(* Logix 5000 project; controller P2 vendor 1 type 14 code 92 rev 20.55; software revision 20.01 *)

TASK MainTask (continuous, watchdog 500 ms) : MainProgram

MODULES
   Local : vendor 1 type 14 code 92 (ICP 0, rev 20.55)
      P2_EN2T_PCN : 1756-EN2T (ICP 1, Ethernet 192.168.1.20, rev 10.1)
         P5 : 1756-EN2T (Ethernet 192.168.1.50, rev 10.1, Output RPI 10 ms)
            P5_CONTROLLER : vendor 1 type 14 code 92 (ICP 0, rev 20.1)
         P4 : 1756-EN2T (Ethernet 192.168.1.40, rev 10.1, Output RPI 10 ms)
            P4_CONTROLLER : vendor 1 type 14 code 92 (ICP 0, rev 20.1)
         P3 : 1756-EN2T (Ethernet 192.168.1.30, rev 10.1, Output RPI 10 ms)
            P3_CONTROLLER : vendor 1 type 14 code 92 (ICP 0, rev 20.1)
      P2_EN2TR_RIO : vendor 1 type 12 code 200 (ICP 2, Ethernet 192.168.0.20, rev 10.1)
         RIO2 : 1794-AENTR (Ethernet 192.168.0.22, rev 1.1, Output RPI 20 ms)
            RIO2_DI : 1794-IB32 (Flex 0, rev 1.1, Input RPI 20 ms)
            RIO2_DO : vendor 1 type 7 code 35 (Flex 1, rev 1.1)
            RIO2_AI : 1794-IE12 (Flex 2, rev 1.1, Output RPI 80 ms)
         WRIO2 : vendor 309 type 12 code 1000 (Ethernet 192.168.0.25, rev 3.1, Output RPI 20 ms)
            WRIO2_AI : 1734-IE4C (PointIO 1, rev 3.1, Input RPI 80 ms)
END_MODULES

TYPE AIN_UDT :
STRUCT
   Pv : REAL;
   Heu : REAL;
   Leu : REAL;
   SAHH : REAL;
   SAH : REAL;
   SAL : REAL;
   SALL : REAL;
   AHH : BOOL;
   AH : BOOL;
   AL : BOOL;
   ALL : BOOL;
   Wifi_Enb : BOOL;
   Hty : BOOL;
   Sim : BOOL;
   Sim_PV : REAL;
END_STRUCT
END_TYPE

TYPE AUTOINP_UDT :
STRUCT
   ON : BOOL;
END_STRUCT
END_TYPE

TYPE ControllerLEDStatus :
STRUCT
   Off : BOOL;
   SolidGreen : BOOL;
   FlashingGreen : BOOL;
   SolidYellow : BOOL;
   FlashingYellow : BOOL;
   FlashingRed : BOOL;
   SolidRed : BOOL;
END_STRUCT
END_TYPE

TYPE DOSING_SETPOINT_UDT :
STRUCT
   High_Setpoint : REAL;
   Low_Setpoint : REAL;
END_STRUCT
END_TYPE

TYPE Duty2_UDT :
STRUCT
   Selection : INT;
   Pmp1_Not_Avl : BOOL;
   Pmp2_Not_Avl : BOOL;
   Selected_Pmp_Not_Avl : BOOL;
   Both_Pmp_Not_Avl : BOOL;
END_STRUCT
END_TYPE

TYPE FaultRecord :
STRUCT
   timelow : DINT;
   timehigh : DINT;
   type : INT;
   code : INT;
   info : DINT[8];
END_STRUCT
END_TYPE

TYPE FIT_UDT :
STRUCT
   Pv : REAL;
   Heu : REAL;
   Leu : REAL;
   SAHH : REAL;
   SAH : REAL;
   SAL : REAL;
   SALL : REAL;
   Totaliser : REAL;
   AHH : BOOL;
   AH : BOOL;
   AL : BOOL;
   ALL : BOOL;
   Sim : BOOL;
   Sim_PV : REAL;
   Wifi_Enb : BOOL;
   Rst_Totaliser : BOOL;
   Hty : BOOL;
END_STRUCT
END_TYPE

TYPE Logix_Status_FP :
STRUCT
   ClearMinorFaults : DINT;
   Sts_MinorFaultEvents : DINT;
   Sts_MinorFaultBits : DINT;
   Sts_Redundant : DINT;
   Set_FaceplateAnimation : DINT;
   Val_ProductCode : DINT;
   MemoryTemp : INT[29];
   Val_raw_data : INT;
   Sts_IO_LED_raw : INT;
   Sts_ProductCode : INT;
   Val_Force_data_raw : INT;
   MemoryRequestData : SINT[12];
   Sts_Force_Installed : BOOL;
   Sts_Force_Enabled : BOOL;
   Sts_Faulted : BOOL;
   Sts_Run : BOOL;
   Sts_Program : BOOL;
   Sts_Minor_fault : BOOL;
   Sts_Major_fault : BOOL;
   Sts_KS_in_run : BOOL;
   Sts_KS_in_program : BOOL;
   Sts_KS_in_remote : BOOL;
   Sts_Changingmodes : BOOL;
   Sts_Test : BOOL;
   Sts_Ladder_Working : BOOL;
   Cmd_ClearFaultRecord : BOOL;
   Set_Controller_Description : STRING;
   UpdateDelayTimer : TIMER;
   Val_MajorFault : FaultRecord;
   Val_MFS : FaultRecord;
   Sts_IO_LED : ControllerLEDStatus;
   Sts_Battery_LED : ControllerLEDStatus;
   MemoryData : Memory_Data;
   TEST : DINT;
END_STRUCT
END_TYPE

TYPE Memory_Data :
STRUCT
   Free_Mem_IO : DINT;
   Free_Mem_DT : DINT;
   Free_Memory : DINT;
   Total_Mem_IO : DINT;
   Total_Mem_DT : DINT;
   Total_Memory : DINT;
   Biggest_IO_Mem_Size_Ava : DINT;
   Biggest_DT_Mem_Size_Ava : DINT;
END_STRUCT
END_TYPE

TYPE MV_UDT :
STRUCT
   Cmd : INT;
   Status : INT;
   Reset : BOOL;
   Auto : BOOL;
   FTO : BOOL;
   FTC : BOOL;
   Avl : BOOL;
END_STRUCT
END_TYPE

TYPE PLANT_AUTO_UDT :
STRUCT
   ON : BOOL;
   OFF : BOOL;
END_STRUCT
END_TYPE

TYPE PLANT_UDT :
STRUCT
   START : BOOL;
   STOP : BOOL;
END_STRUCT
END_TYPE

TYPE PMP_UDT :
STRUCT
   Cmd : INT;
   Status : INT;
   RunMin : REAL;
   Total_RunMin : REAL;
   RunHr : REAL;
   Total_RunHr : REAL;
   Remote : BOOL;
   Auto : BOOL;
   Fault : BOOL;
   Avl : BOOL;
   Permissive : DINT;
   Shutdown : DINT;
   SD : DINT;
   Reset : BOOL;
   Reset_RunHr : BOOL;
   FTR : BOOL;
   FTS : BOOL;
END_STRUCT
END_TYPE

TYPE PRECONDITION_UDT :
STRUCT
   PERMISSIVE1 : BOOL;
   PERMISSIVE2 : BOOL;
   PERMISSIVE3 : BOOL;
   PERMISSIVE4 : BOOL;
   PERMISSIVE5 : BOOL;
   SHUTDOWN1 : BOOL;
   SHUTDOWN2 : BOOL;
   SHUTDOWN3 : BOOL;
   SHUTDOWN4 : BOOL;
   SHUTDOWN5 : BOOL;
END_STRUCT
END_TYPE

TYPE RED_STAT :
STRUCT
   Redundancy_status_of_the_controller : INT;
   Redundancy_state_of_the_partner : INT;
END_STRUCT
END_TYPE

TYPE SWITCH_UDT :
STRUCT
   Alarm : BOOL;
   Delay : DINT;
END_STRUCT
END_TYPE

TYPE WIFI_UDT :
STRUCT
   PLC_WIFI : BOOL;
   RIO_WIFI : BOOL;
END_STRUCT
END_TYPE

ADD_ON_INSTRUCTION AIN_FBD   (* revision 1.0 *)
VAR_INPUT
   WRIO_Enb : BOOL; {visible}
   Raw_RIO : INT; {visible}
   Raw_WRIO : INT; {visible}
   L_Raw_RIO : INT; {visible}
   H_Raw_RIO : INT; {visible}
   L_Raw_WRIO : INT; {visible}
   H_Raw_WRIO : INT; {visible}
   HEU : INT; {visible}
   LEU : INT; {visible}
END_VAR
VAR_OUTPUT
   Hty : BOOL; {visible}
   Wifi_Enb : BOOL; {access Read Only, visible}
   AHH : BOOL; {visible}
   AH : BOOL; {access Read Only, visible}
   AL : BOOL; {access Read Only, visible}
   ALL : BOOL; {visible}
END_VAR
VAR_INPUT
   SAHH : REAL; {visible}
   SAH : REAL; {visible}
   SAL : REAL; {visible}
   SALL : REAL; {visible}
   Simulation : BOOL; {visible}
   RIO_Hty : BOOL; {visible}
   WRIO_Hty : BOOL; {visible}
END_VAR
VAR_IN_OUT
   Pv : REAL; {required}
   Sim_PV : REAL; {required}
   HMI : AIN_UDT; {required}
END_VAR
VAR
   SCALE : SCALE; {access None}
   ALM : ALARM; {access None}
   _Raw : INT; {access None}
   _L_Raw : INT; {access None}
   _H_Raw : INT; {access None}
   _Inst_Hty : BOOL; {access None}
END_VAR

ROUTINE Logic   (* structured text *)
   (*RIO and Wireless RIO Selection*)
   
   IF WRIO_Enb THEN
   	Wifi_Enb	:= 1;
   	_Raw		:= Raw_WRIO;
   	_H_Raw		:= H_Raw_WRIO;
   	_L_Raw		:= L_Raw_WRIO;
   	_Inst_Hty 	:= WRIO_Hty;
   ELSE
   	Wifi_Enb	:= 0;
   	_Raw		:= Raw_RIO;
   	_H_Raw		:= H_Raw_RIO;
   	_L_Raw		:= L_Raw_RIO;
   	_Inst_Hty 	:= RIO_Hty;
   END_IF;
   
   (*Calculation for PV*)
   IF Simulation THEN
   	Pv	:=Sim_PV;
   ELSE
   	SCALE.In		:=_Raw;
   	SCALE.InRawMax	:=_H_Raw;
   	SCALE.InRawMin	:=_L_Raw;
   	SCALE.InEUMax	:=HEU;
   	SCALE.InEUMin	:=LEU;
   	SCL(SCALE);
   
   	IF SCALE.Out<0 THEN
   		Pv	:= 0.0;
   	ELSE
   		Pv	:=SCALE.Out;
   	END_IF;
   
   	Sim_PV	:=Pv;
   
   END_IF;
   
   (*Alarms*)
   ALM.In			:=Pv;
   ALM.HHLimit		:=SAHH;
   ALM.HLimit		:=SAH;
   ALM.LLimit		:=SAL;
   ALM.LLLimit		:=SALL;
   ALM(ALM);
   
   AHH				:=ALM.HHAlarm;
   AH				:=ALM.HAlarm;
   AL				:=ALM.LAlarm;
   ALL				:=ALM.LLAlarm;
   
   Hty:= _Inst_Hty AND (_Raw > _L_Raw) AND (_Raw < _H_Raw)  ;
   
   
   
   
   
   
END_ROUTINE
END_ADD_ON_INSTRUCTION

ADD_ON_INSTRUCTION Duty2_FBD   (* revision 1.0 *)
VAR_INPUT
   AutoInp : BOOL; {visible}
   Selection : INT; {visible}
   Pmp1_Avl : BOOL; {visible}
   Pmp2_Avl : BOOL; {visible}
END_VAR
VAR_OUTPUT
   Start_Pmp1 : BOOL; {visible}
   Start_Pmp2 : BOOL; {visible}
END_VAR
VAR_IN_OUT
   HMI : Duty2_UDT; {required}
END_VAR

ROUTINE Logic   (* structured text *)
   IF AutoInp THEN
   	CASE Selection OF
   		(*PUMP 1 *)
   		1:
   			IF Pmp1_Avl THEN
   				Start_Pmp1					:=1;
   				Start_Pmp2					:=0;
   				HMI.Selected_Pmp_Not_Avl	:=0;
   			ELSIF NOT Pmp1_Avl AND Pmp2_Avl THEN
   				Start_Pmp1					:=0;
   				Start_Pmp2					:=1;
   				HMI.Selected_Pmp_Not_Avl	:=1;
   			ELSIF NOT Pmp1_Avl AND NOT Pmp2_Avl	THEN
   				Start_Pmp1					:=0;
   				Start_Pmp2					:=0;
   			END_IF;
   
   		(*PUMP 2 *)
   		2:
   			IF Pmp2_Avl THEN
   				Start_Pmp1					:=0;
   				Start_Pmp2					:=1;
   				HMI.Selected_Pmp_Not_Avl	:=0;
   			ELSIF NOT Pmp2_Avl AND Pmp1_Avl THEN
   				Start_Pmp1					:=1;
   				Start_Pmp2					:=0;
   				HMI.Selected_Pmp_Not_Avl	:=1;
   			ELSIF NOT Pmp1_Avl AND NOT Pmp2_Avl	THEN
   				Start_Pmp1					:=0;
   				Start_Pmp2					:=0;
   			END_IF;
   	END_CASE;
   ELSE
   	Start_Pmp1					:=0;
   	Start_Pmp2					:=0;
   END_IF;
   
   
END_ROUTINE
END_ADD_ON_INSTRUCTION

ADD_ON_INSTRUCTION FIT_FBD   (* revision 1.0 *)
VAR_INPUT
   WRIO_Enb : BOOL; {visible}
   Raw_RIO : INT; {visible}
   Raw_WRIO : INT; {visible}
   L_Raw_RIO : INT; {visible}
   H_Raw_RIO : INT; {visible}
   L_Raw_WRIO : INT; {visible}
   H_Raw_WRIO : INT; {visible}
   HEU : REAL; {visible}
   LEU : REAL; {visible}
END_VAR
VAR_OUTPUT
   Hty : BOOL; {visible}
   Wifi_Enb : BOOL; {visible}
   AHH : BOOL; {visible}
   AH : BOOL; {access Read Only, visible}
   AL : BOOL; {access Read Only, visible}
   ALL : BOOL; {visible}
END_VAR
VAR_INPUT
   SAHH : REAL; {visible}
   SAH : REAL; {visible}
   SAL : REAL; {visible}
   SALL : REAL; {visible}
   Simulation : BOOL; {visible}
   RIO_Hty : BOOL; {visible}
   WRIO_Hty : BOOL; {visible}
   Totaliser_Enb : BOOL; {visible}
   Rst_Totaliser : BOOL; {visible}
END_VAR
VAR_IN_OUT
   Totaliser : REAL; {required}
   Pv : REAL; {required}
   Sim_Pv : REAL; {required}
   HMI : FIT_UDT; {required}
END_VAR
VAR
   SCALE : SCALE; {access None}
   ALM : ALARM; {access None}
   TON : FBD_TIMER; {access None}
   _SEC_P : BOOL; {access None}
   _Inst_Hty : BOOL; {access None}
   _L_Raw : INT; {access None}
   _H_Raw : INT; {access None}
   _Raw : INT; {access None}
   R_TRIG : FBD_ONESHOT; {access None}
END_VAR

ROUTINE Logic   (* structured text *)
   (*RIO and Wireless RIO Selection*)
   
   IF WRIO_Enb THEN
   	Wifi_Enb	:= 1;
   	_Raw		:= Raw_WRIO;
   	_H_Raw		:= H_Raw_WRIO;
   	_L_Raw		:= L_Raw_WRIO;
   	_Inst_Hty 	:= WRIO_Hty;
   ELSE
   	Wifi_Enb	:= 0;
   	_Raw		:= Raw_RIO;
   	_H_Raw		:= H_Raw_RIO;
   	_L_Raw		:= L_Raw_RIO;
   	_Inst_Hty 	:= RIO_Hty;
   END_IF;
   
   (*Calculation for PV*)
   IF Simulation THEN
   	Pv	:= Sim_Pv   ;
   ELSE
   	SCALE.In		:=_Raw;
   	SCALE.InRawMax	:=_H_Raw;
   	SCALE.InRawMin	:=_L_Raw;
   	SCALE.InEUMax	:=HEU;
   	SCALE.InEUMin	:=LEU;
   	SCL(SCALE);
   	IF SCALE.Out>0 THEN
   		Pv	:=SCALE.Out;
   	ELSIF SCALE.Out<=0 THEN
   		Pv	:=0.0;
   	END_IF;
   
   	Sim_Pv	:=Pv;
   END_IF;
   
   (*Alarms*)
   ALM.In			:=Pv;
   ALM.HHLimit		:=SAHH;
   ALM.HLimit		:=SAH;
   ALM.LLimit		:=SAL;
   ALM.LLLimit		:=SALL;
   ALM(ALM);
   
   AHH				:=ALM.HHAlarm;
   AH				:=ALM.HAlarm;
   AL				:=ALM.LAlarm;
   ALL				:=ALM.LLAlarm;
   
   (*SECOND PULSE*)
   TON.PRE	:=1000;
   TON.TimerEnable	:=1;
   TONR(TON );
   R_TRIG.InputBit :=TON.DN ;
   OSRI( R_TRIG);
   _SEC_P  := R_TRIG.OutputBit;
   TON.Reset := _SEC_P;
   
   IF Totaliser_Enb THEN
   	IF _SEC_P THEN
   		HMI.Totaliser := HMI.Totaliser +  (ABS(Pv) / 3600 );
   	END_IF;
   END_IF;
   
   IF  Rst_Totaliser   THEN
   	HMI.Totaliser	:=0;
   END_IF;
   
   Hty:= _Inst_Hty AND (_Raw > _L_Raw) AND (_Raw < _H_Raw)  ;
   
   
   
   
   
   
END_ROUTINE
END_ADD_ON_INSTRUCTION

ADD_ON_INSTRUCTION MV_FBD   (* revision 1.0 *)
VAR_INPUT
   Auto : BOOL; {visible}
END_VAR
VAR_OUTPUT
   Cmd_Open : BOOL; {visible}
   Cmd_Close : BOOL; {visible}
   FTO : BOOL; {visible}
   FTC : BOOL; {access Read Only, visible}
END_VAR
VAR_INPUT
   AutoInp : BOOL; {visible}
   ZSO : BOOL; {visible}
   Open_TM : DINT; {visible}
   ZSC : BOOL; {visible}
   Close_TM : DINT; {visible}
END_VAR
VAR_IN_OUT
   Cmd : INT; {required}
   HMI : MV_UDT; {required}
END_VAR
VAR
   TON_Open_TM : FBD_TIMER; {access None}
   TON_Close_TM : FBD_TIMER; {access None}
END_VAR

ROUTINE Logic   (* structured text *)
   (*Fail to Close*)
   TON_Close_TM.PRE 			:= 	Close_TM*1000;
   TON_Close_TM.TimerEnable 	:=  Cmd_Close;
   TONR(TON_Close_TM);
   
   (*Fail to Open*)
   TON_Open_TM.PRE 			:= 	Open_TM*1000;
   TON_Open_TM.TimerEnable 	:= 	Cmd_Open;
   TONR(TON_Open_TM);
   
   IF ZSC THEN
   	HMI.Status	:=1;
   ELSIF ZSO THEN
   	HMI.Status	:=2;
   ELSE
   	HMI.Status	:=0;
   END_IF;
   
   HMI.Avl:= Auto AND NOT FTC AND NOT FTO;
   
   IF HMI.Reset THEN
   	(*IF NOT TON_Close_TM.DN AND ZSC THEN*)
   			FTC		:= 0;
   	(*END_IF;*)
   	(*IF NOT TON_Open_TM.DN AND ZSO THEN*)
   			FTO		:= 0;
   	(*END_IF;*)
   END_IF;
   
   IF  NOT Auto THEN
   	CASE HMI.Cmd OF
   		1:	(*CLOSE*)
   			Cmd_Close	:= 1;
   			Cmd_Open	:= 0;
   			IF TON_Close_TM.DN AND (NOT ZSC) THEN
   				FTC		:= 1;
   				FTO		:= 0;
   			END_IF;
   		2:	(*OPEN*)
   			IF FTO OR FTC    THEN
   				HMI.Cmd := 1;
   			END_IF;
   
   			IF NOT FTC AND NOT FTO THEN
   				Cmd_Close	:= 0;
   				Cmd_Open	:= 1;
   			END_IF;
   
   			IF TON_Open_TM.DN AND (NOT ZSO) THEN
   				FTC		:= 0;
   				FTO		:= 1;
   				HMI.Cmd := 1;
   			END_IF;
   	END_CASE;
   ELSE
   	(*Maintain Last status when switching from Auto to Manual*)
   	IF ZSO THEN
   		Cmd	:= 2;
   	END_IF;
   	IF ZSC THEN
   		Cmd	:= 1;
   	END_IF;
   
   	IF  AutoInp AND (NOT FTC AND NOT FTO) THEN
   		Cmd_Close	:= 0;
   		Cmd_Open	:= 1;
   		IF TON_Open_TM.DN AND (NOT ZSO) THEN
   			FTC		:= 0;
   			FTO		:= 1;
   		END_IF;
   	ELSE
   		Cmd_Close	:= 1;
   		Cmd_Open	:= 0;
   		IF TON_Close_TM.DN AND (NOT ZSC) THEN
   			FTC		:= 1;
   			FTO		:= 0;
   		END_IF;
   	END_IF;
   END_IF;
   
   
END_ROUTINE
END_ADD_ON_INSTRUCTION

ADD_ON_INSTRUCTION PMP_FBD   (* revision 1.0 *)
VAR_OUTPUT
   Cmd_Start : BOOL; {visible}
   Avl : BOOL; {visible}
   Fault : BOOL; {visible}
   FT_Stop : BOOL; {visible}
   FT_Start : BOOL; {visible}
   RunHr : REAL; {visible}
   Total_RunHr : REAL; {visible}
   SD : DINT; {access Read Only, visible}
END_VAR
VAR_INPUT
   Auto : BOOL; {visible}
   AutoInp : BOOL; {visible}
   Remote : BOOL; {visible}
   Run : BOOL; {visible}
   Trip : BOOL; {visible}
   Start_TM : DINT; {visible}
   Stop_TM : DINT; {visible}
   Rst : BOOL; {visible}
   Rst_RunHr : BOOL; {visible}
   Permissive : DINT; {visible}
   Shutdown : DINT; {visible}
END_VAR
VAR_IN_OUT
   RunMin : REAL; {required}
   Total_RunMin : REAL; {required}
   Cmd : INT; {required}
   HMI : PMP_UDT; {required}
END_VAR
VAR
   TON_Start_TM : FBD_TIMER; {access None}
   TON_Stop_TM : FBD_TIMER; {access None}
   _Min_P : BOOL; {access None}
   TON_Min : FBD_TIMER; {access None}
   R_TRIG_SEC : FBD_ONESHOT; {access None}
END_VAR

ROUTINE Logic   (* structured text *)
   (*Fail to Start*)
   TON_Start_TM.PRE 			:= 	Start_TM*1000;
   TON_Start_TM.TimerEnable 	:=  Cmd_Start;
   TONR(TON_Start_TM);
   
   (*Fail to Stop*)
   TON_Stop_TM.PRE 			:= 	Stop_TM*1000;
   TON_Stop_TM.TimerEnable 	:=  NOT Cmd_Start;
   TONR(TON_Stop_TM);
   
   IF (NOT Run) THEN
   	HMI.Status	:=1;
   ELSE
   	HMI.Status	:=2;
   END_IF;
   
   IF Fault THEN
   	HMI.Fault:= 1;
   ELSE
   	HMI.Fault:= 0;
   END_IF;
   
   IF HMI.Reset THEN
   	IF NOT TON_Stop_TM.DN THEN
   			FT_Stop		:= 0;
   	END_IF;
   	IF NOT TON_Start_TM.DN THEN
   			FT_Start	:= 0;
   	END_IF;
   
   	SD :=0;
   
   END_IF;
   
   Fault		:=Trip OR SD<>0;
   HMI.Remote	:=Remote;
   Avl:= Auto AND Remote AND NOT Fault AND NOT FT_Start AND NOT FT_Stop AND SD=0 ;
   
   IF Remote THEN
   	IF  NOT Auto THEN
   		CASE HMI.Cmd OF
   			1:	(*Stop*)
   				Cmd_Start	:=0;
   				IF TON_Stop_TM.DN AND Run THEN
   					FT_Start	:= 0;
   					FT_Stop		:= 1;
   				END_IF;
   			2:	(*OPEN*)
   				IF NOT Fault AND NOT FT_Start AND NOT FT_Stop AND (Permissive=-1) AND HMI.SD=0 THEN
   					Cmd_Start	:= 1;
   				ELSIF Cmd_Start AND (HMI.SD<>0) OR Fault THEN
   					SD				:= HMI.SD;
   					Cmd_Start		:= 0;
   					HMI.Cmd 		:= 1;
   				ELSIF (Permissive<>-1) THEN
   					HMI.Cmd 		:= 1;
   				END_IF;
   
   				IF TON_Start_TM.DN AND NOT Run THEN
   					FT_Start	:= 1;
   					FT_Stop		:= 0;
   					Cmd_Start	:= 0;
   					HMI.Cmd 	:= 1;
   				END_IF;
   		END_CASE;
   	ELSE
   		IF Run THEN
   			Cmd	:= 2;
   		END_IF;
   		IF (NOT Run) OR Fault OR FT_Start OR FT_Stop THEN
   			Cmd	:= 1;
   		END_IF;
   
   		IF  AutoInp  THEN
   			IF NOT Fault AND NOT FT_Start AND NOT FT_Stop AND (Permissive=-1) AND HMI.SD=0  THEN
   				Cmd_Start	:=1;
   			ELSIF Cmd_Start OR (HMI.SD<>0) OR Fault THEN
   				SD			:= HMI.SD;
   				Cmd_Start	:=0;
   			END_IF;
   
   			IF TON_Start_TM.DN AND NOT Run THEN
   				FT_Start	:= 1;
   				FT_Stop		:= 0;
   				Cmd_Start	:= 0;
   				HMI.Cmd 	:= 1;
   			END_IF;
   		ELSE
   			Cmd_Start	:=0;
   			IF TON_Stop_TM.DN AND Run THEN
   				FT_Start	:= 0;
   				FT_Stop		:= 1;
   
   			END_IF;
   		END_IF;
   	END_IF;
   
   ELSE (*Local*)
   	Cmd_Start	:=0;
   	Cmd	:= 1;
   
   	FT_Start	:= 0;
   	FT_Stop		:= 0;
   
   
   
   
   	(*	IF Run THEN
   			Cmd	:= 2;
   		END_IF;
   		IF (NOT Run) OR Fault OR FT_Start OR FT_Stop THEN
   			Cmd	:= 1;
   		END_IF;
   		*)
   END_IF;
   
   (*1 MIN PULSE*)
   TON_Min.PRE	:=60000;
   TON_Min.TimerEnable	:=1;
   TONR(TON_Min );
   R_TRIG_SEC.InputBit :=TON_Min.DN ;
   OSRI( R_TRIG_SEC);
   _Min_P  := R_TRIG_SEC.OutputBit;
   TON_Min.Reset 	:= _Min_P;
   
   IF Run THEN
   	IF _Min_P THEN
   		RunMin 			:=RunMin + 1.0;
   		Total_RunMin	:=Total_RunMin + 1.0;
   	END_IF;
   END_IF;
   
   RunHr 				:=RunMin/60.0;
   Total_RunHr			:=Total_RunMin/60.0;
   
   IF  Rst_RunHr THEN
   	RunMin	:=0;
   END_IF;
   
   
   
END_ROUTINE
END_ADD_ON_INSTRUCTION

ADD_ON_INSTRUCTION SWITCH_FBD   (* revision 1.0 *)
VAR_INPUT
   Alarm : BOOL; {visible}
   Delay : DINT; {required}
END_VAR
VAR_OUTPUT
   Status : BOOL; {access None, required}
END_VAR
VAR_IN_OUT
   HMI : SWITCH_UDT; {required}
END_VAR
VAR
   TON_Delay_Sec : FBD_TIMER; {access None}
END_VAR

ROUTINE Logic   (* structured text *)
   (*Delay for Alarm*)
   TON_Delay_Sec.PRE 			:= 	Delay*1000;
   TON_Delay_Sec.TimerEnable 	:=  Alarm;
   TONR(TON_Delay_Sec);
   
   Status := TON_Delay_Sec.DN ;
END_ROUTINE
END_ADD_ON_INSTRUCTION

VAR_GLOBAL   (* controller tags *)
   _FIT201_Tot_Enb : BOOL := 1;
   _MV201_AutoInp : BOOL := 1;
   _MV201_AutoInp_P1 : INT;
   _P201_AutoInp : BOOL;
   _P202_AutoInp : BOOL;
   _P203_AutoInp : BOOL := 1;
   _P204_AutoInp : BOOL;
   _P205_AutoInp : BOOL := 1;
   _P206_AutoInp : BOOL;
   _P207_AutoInp : BOOL;
   _P208_AutoInp : BOOL;
   _P_HCL_DUTY_AutoInp : BOOL := 1;
   _P_NACL_DUTY_AutoInp : BOOL;
   _P_NAOCL_FAC_DUTY_AutoInp : BOOL := 1;
   _P_NAOCL_UF_DUTY_AutoInp : BOOL;
   _P_RAW_WATER_DUTY_AutoInp : BOOL;
   AI_AIT_201_COND : INT := 6270;
   AI_AIT_201_COND_HTY : BOOL := 1;
   AI_AIT_202_PH : INT := 21186;
   AI_AIT_202_PH_HTY : BOOL := 1;
   AI_AIT_203_ORP : INT := 15913;
   AI_AIT_203_ORP_HTY : BOOL := 1;
   AI_FIT_201_FLOW : INT := -11;
   AI_FIT_201_FLOW_HTY : BOOL := 1;
   AI_RIO2_SPARE_03 : INT;
   AI_RIO2_SPARE_03_HTY : BOOL;
   AI_RIO2_SPARE_04 : INT := -7699;
   AI_RIO2_SPARE_04_HTY : BOOL := 1;
   AI_RIO2_SPARE_05 : INT := -7701;
   AI_RIO2_SPARE_05_HTY : BOOL := 1;
   AI_RIO2_SPARE_06 : INT := -7701;
   AI_RIO2_SPARE_06_HTY : BOOL := 1;
   AI_RIO2_SPARE_07 : INT := -7700;
   AI_RIO2_SPARE_07_HTY : BOOL := 1;
   AI_RIO2_SPARE_08 : INT := -7700;
   AI_RIO2_SPARE_08_HTY : BOOL := 1;
   AI_RIO2_SPARE_09 : INT := -7703;
   AI_RIO2_SPARE_09_HTY : BOOL := 1;
   AI_RIO2_SPARE_10 : INT := -7700;
   AI_RIO2_SPARE_10_HTY : BOOL := 1;
   AI_RIO2_SPARE_11 : INT := -7700;
   AI_RIO2_SPARE_11_HTY : BOOL := 1;
   AIT201_FB : AIN_FBD := (Raw_RIO := 6270, Raw_WRIO := 16743, H_Raw_RIO := 31208, L_Raw_WRIO := 3277, H_Raw_WRIO := 16383, HEU := 1000, Hty := 1, AL := 1, SAHH := 950.0, SAH := 260.0, SAL := 250.0, SALL := 50.0, RIO_Hty := 1);
   AIT202_FB : AIN_FBD := (Raw_RIO := 21186, Raw_WRIO := 11550, H_Raw_RIO := 31208, L_Raw_WRIO := 3277, H_Raw_WRIO := 16383, HEU := 12, LEU := 2, Hty := 1, AH := 1, SAHH := 12.0, SAH := 7.05, SAL := 6.95, SALL := 3.0, RIO_Hty := 1, WRIO_Hty := 1);
   AIT203_FB : AIN_FBD := (Raw_RIO := 15909, Raw_WRIO := 7064, H_Raw_RIO := 31208, L_Raw_WRIO := 3277, H_Raw_WRIO := 16383, HEU := 800, Hty := 1, AL := 1, SAHH := 750.0, SAH := 480.0, SAL := 440.0, SALL := 100.0, RIO_Hty := 1, WRIO_Hty := 1);
   DI_LS_201_LOW : BOOL;
   DI_LS_202_LOW : BOOL;
   DI_LS_203_LOW : BOOL;
   DI_LS_203_LOWLOW : BOOL;
   DI_MV_201_ZSC : BOOL;
   DI_MV_201_ZSO : BOOL := 1;
   DI_P_201_AUTO : BOOL := 1;
   DI_P_201_FAULT : BOOL;
   DI_P_201_RUN : BOOL;
   DI_P_202_AUTO : BOOL := 1;
   DI_P_202_FAULT : BOOL;
   DI_P_202_RUN : BOOL;
   DI_P_203_AUTO : BOOL := 1;
   DI_P_203_FAULT : BOOL;
   DI_P_203_RUN : BOOL;
   DI_P_204_AUTO : BOOL := 1;
   DI_P_204_FAULT : BOOL;
   DI_P_204_RUN : BOOL;
   DI_P_205_AUTO : BOOL := 1;
   DI_P_205_FAULT : BOOL;
   DI_P_205_RUN : BOOL;
   DI_P_206_AUTO : BOOL := 1;
   DI_P_206_FAULT : BOOL;
   DI_P_206_RUN : BOOL;
   DI_P_207_AUTO : BOOL := 1;
   DI_P_207_FAULT : BOOL;
   DI_P_207_RUN : BOOL;
   DI_P_208_AUTO : BOOL := 1;
   DI_P_208_FAULT : BOOL;
   DI_P_208_RUN : BOOL;
   DI_WIFI_PLC_2 : BOOL;
   DI_WIFI_RIO_2 : BOOL;
   DO_MV_201_CLOSE : BOOL;
   DO_MV_201_OPEN : BOOL := 1;
   DO_P_201_START : BOOL;
   DO_P_202_START : BOOL;
   DO_P_203_START : BOOL;
   DO_P_204_START : BOOL;
   DO_P_205_START : BOOL;
   DO_P_206_START : BOOL;
   DO_P_207_START : BOOL;
   DO_P_208_START : BOOL;
   DO_RIO2_SPARE_04 : BOOL;
   DO_RIO2_SPARE_05 : BOOL;
   DO_RIO2_SPARE_06 : BOOL;
   DO_RIO2_SPARE_07 : BOOL;
   DO_RIO2_SPARE_08 : BOOL;
   DO_RIO2_SPARE_09 : BOOL;
   DO_RIO2_SPARE_10 : BOOL;
   DO_RIO2_SPARE_11 : BOOL;
   DO_RIO2_SPARE_12 : BOOL;
   DO_RIO2_SPARE_13 : BOOL;
   DO_RIO2_SPARE_14 : BOOL;
   DO_RIO2_SPARE_15 : BOOL;
   FIT201_FB : FIT_FBD := (Raw_RIO := -11, Raw_WRIO := 3263, L_Raw_RIO := -5, H_Raw_RIO := 31208, L_Raw_WRIO := 3277, H_Raw_WRIO := 16383, HEU := 4.0, AL := 1, ALL := 1, SAHH := 3.5, SAH := 2.0, RIO_Hty := 1, WRIO_Hty := 1, Totaliser_Enb := 1);
   HMI_AIT201 : AIN_UDT := (Pv := 200.91002, SAHH := 950.0, SAH := 260.0, SAL := 250.0, SALL := 50.0, AL := 1, Hty := 1, Sim_PV := 200.91002);
   HMI_AIT202 : AIN_UDT := (Pv := 8.788645, SAHH := 12.0, SAH := 7.05, SAL := 6.95, SALL := 3.0, AH := 1, Hty := 1, Sim_PV := 8.788645);
   HMI_AIT203 : AIN_UDT := (Pv := 407.76724, SAHH := 750.0, SAH := 480.0, SAL := 440.0, SALL := 100.0, AL := 1, Hty := 1, Sim_PV := 407.76724);
   HMI_AIT402 : AIN_UDT := (Pv := 249.7052, SAHH := 800.0, SAH := 300.0, SAL := 250.0, SALL := 200.0, AL := 1, Hty := 1, Sim_PV := 249.7052);
   HMI_AIT501 : AIN_UDT := (Pv := 7.011215, SAHH := 12.0, SAH := 8.0, SAL := 6.0, SALL := 4.0, Hty := 1, Sim_PV := 7.011215);
   HMI_AIT502 : AIN_UDT := (Pv := 175.57037, SAHH := 300.0, SAH := 250.0, Hty := 1, Sim_PV := 175.57037);
   HMI_AIT503 : AIN_UDT := (Pv := 273.26328, SAHH := 500.0, SAH := 260.0, SAL := 250.0, AH := 1, Hty := 1, Sim_PV := 273.26328);
   HMI_AIT504 : AIN_UDT := (Pv := 12.996668, SAHH := 15.0, SAH := 12.0, AH := 1, Hty := 1, Sim_PV := 12.996668);
   HMI_FIT201 : FIT_UDT := (SAHH := 3.5, SAH := 2.0, Totaliser := 30.56272, AL := 1, ALL := 1);
   HMI_HCL_PH_DOSING : DOSING_SETPOINT_UDT;
   HMI_LIT301 : AIN_UDT := (Pv := 844.73535, SAHH := 1200.0, SAH := 1000.0, SAL := 800.0, SALL := 250.0, Hty := 1, Sim_PV := 844.73535);
   HMI_LS201 : SWITCH_UDT;
   HMI_LS202 : SWITCH_UDT;
   HMI_LSL203 : SWITCH_UDT;
   HMI_LSLL203 : SWITCH_UDT;
   HMI_MV201 : MV_UDT := (Cmd := 2, Status := 2, Reset := 1, Auto := 1, Avl := 1);
   HMI_MV301 : MV_UDT := (Cmd := 1, Status := 1, Reset := 1, Auto := 1, Avl := 1);
   HMI_NACL_COND_DOSING : DOSING_SETPOINT_UDT;
   HMI_NAOCL_FAC_FAC_DOSING : DOSING_SETPOINT_UDT;
   HMI_NAOCL_FAC_UF_DOSING : DOSING_SETPOINT_UDT;
   HMI_P201 : PMP_UDT := (Cmd := 1, Status := 1, RunMin := 6385.0, Total_RunMin := 6385.0, RunHr := 106.416664, Total_RunHr := 106.416664, Remote := 1, Auto := 1, Avl := 1, Permissive := -5, Reset := 1);
   HMI_P201_MSG : PRECONDITION_UDT := (PERMISSIVE1 := 1, PERMISSIVE2 := 1);
   HMI_P202 : PMP_UDT := (Cmd := 1, Status := 1, RunMin := 6.0, Total_RunMin := 6.0, RunHr := 0.1, Total_RunHr := 0.1, Remote := 1, Auto := 1, Avl := 1, Permissive := -5, Reset := 1);
   HMI_P202_MSG : PRECONDITION_UDT := (PERMISSIVE1 := 1, PERMISSIVE2 := 1);
   HMI_P203 : PMP_UDT := (Cmd := 1, Status := 1, RunMin := 9688.0, Total_RunMin := 9688.0, RunHr := 161.46666, Total_RunHr := 161.46666, Remote := 1, Auto := 1, Avl := 1, Permissive := -5, Reset := 1);
   HMI_P203_MSG : PRECONDITION_UDT := (PERMISSIVE1 := 1, PERMISSIVE2 := 1);
   HMI_P204 : PMP_UDT := (Cmd := 1, Status := 1, RunMin := 6.0, Total_RunMin := 6.0, RunHr := 0.1, Total_RunHr := 0.1, Remote := 1, Auto := 1, Avl := 1, Permissive := -5, Reset := 1);
   HMI_P204_MSG : PRECONDITION_UDT := (PERMISSIVE1 := 1, PERMISSIVE2 := 1);
   HMI_P205 : PMP_UDT := (Cmd := 1, Status := 1, RunMin := 8631.0, Total_RunMin := 8631.0, RunHr := 143.85, Total_RunHr := 143.85, Remote := 1, Auto := 1, Avl := 1, Permissive := -5, Reset := 1);
   HMI_P205_MSG : PRECONDITION_UDT := (PERMISSIVE1 := 1, PERMISSIVE2 := 1);
   HMI_P206 : PMP_UDT := (Cmd := 1, Status := 1, RunMin := 4.0, Total_RunMin := 4.0, RunHr := 0.06666667, Total_RunHr := 0.06666667, Remote := 1, Auto := 1, Avl := 1, Permissive := -5, Reset := 1);
   HMI_P206_MSG : PRECONDITION_UDT := (PERMISSIVE1 := 1, PERMISSIVE2 := 1);
   HMI_P207 : PMP_UDT := (Cmd := 1, Status := 1, RunMin := 1.0, Total_RunMin := 1.0, RunHr := 0.016666668, Total_RunHr := 0.016666668, Remote := 1, Auto := 1, Avl := 1, Permissive := -3, Reset := 1);
   HMI_P207_MSG : PRECONDITION_UDT := (PERMISSIVE1 := 1, PERMISSIVE3 := 1);
   HMI_P208 : PMP_UDT := (Cmd := 1, Status := 1, RunMin := 1.0, Total_RunMin := 1.0, RunHr := 0.016666668, Total_RunHr := 0.016666668, Remote := 1, Auto := 1, Avl := 1, Permissive := -3, Reset := 1);
   HMI_P208_MSG : PRECONDITION_UDT := (PERMISSIVE1 := 1, PERMISSIVE3 := 1);
   HMI_P2_PERMISSIVE : AUTOINP_UDT := (ON := 1);
   HMI_P2_READY : BOOL := 1;
   HMI_P2_SHUTDOWN : BOOL := 1;
   HMI_P2_STATE : INT := 2;
   HMI_P_HCL_DUTY : Duty2_UDT := (Selection := 1);
   HMI_P_NACL_DUTY : Duty2_UDT := (Selection := 1);
   HMI_P_NAOCL_FAC_DUTY : Duty2_UDT := (Selection := 1);
   HMI_P_NAOCL_UF_DUTY : Duty2_UDT := (Selection := 2);
   HMI_P_RAW_WATER_DUTY : Duty2_UDT;
   HMI_PLANT : PLANT_UDT;
   HMI_PLANT_AUTO : PLANT_AUTO_UDT;
   HMI_PLANT_RESET : PLANT_AUTO_UDT;
   HMI_START_PLANT : BOOL;
   HMI_STOP_PLANT : BOOL;
   HMI_WIFI : WIFI_UDT;
   Logix_Status : Logix_Status_FP := (Set_FaceplateAnimation := 90, Val_ProductCode := 92, MemoryTemp[0] := 5, MemoryTemp[1] := 1, MemoryTemp[3] := 29356, MemoryTemp[4] := 3, MemoryTemp[5] := 9148, MemoryTemp[6] := 7, MemoryTemp[9] := 2, MemoryTemp[11] := -4608, MemoryTemp[12] := 3, MemoryTemp[14] := 8, MemoryTemp[17] := 5, MemoryTemp[21] := 6, MemoryTemp[23] := 27326, MemoryTemp[24] := 3, MemoryTemp[25] := 7, MemoryTemp[27] := 8862, MemoryTemp[28] := 7, Val_raw_data := 12384, Sts_IO_LED_raw := 2, Sts_ProductCode := 92, MemoryRequestData[0] := 5, MemoryRequestData[2] := 1, MemoryRequestData[4] := 2, MemoryRequestData[6] := 5, MemoryRequestData[8] := 6, MemoryRequestData[10] := 7, Sts_Run := 1, Sts_KS_in_remote := 1, Sts_Ladder_Working := 1, Set_Controller_Description := 'P2: Pre-Treatment System', UpdateDelayTimer.PRE := 1000, UpdateDelayTimer.ACC := 66, UpdateDelayTimer.EN := 1, UpdateDelayTimer.TT := 1, Val_MFS.timelow := 71751885, Val_MFS.timehigh := 206334, Val_MFS.type := 3, Val_MFS.code := 20, Val_MFS.info[1] := 1, Sts_IO_LED.FlashingGreen := 1, Sts_Battery_LED.Off := 1, MemoryData.Free_Mem_IO := 903856, MemoryData.Free_Mem_DT := 1871600, MemoryData.Total_Mem_IO := 1030144, MemoryData.Total_Mem_DT := 2097152, MemoryData.Biggest_IO_Mem_Size_Ava := 895736, MemoryData.Biggest_DT_Mem_Size_Ava := 1870456);
   LS201_FB : SWITCH_FBD;
   LS202_FB : SWITCH_FBD;
   LS203_FB : SWITCH_FBD;
   LS203_FB_01 : SWITCH_FBD;
   LSLL203_FB : SWITCH_FBD;
   Memory_Message : MESSAGE;
        MessageParameters(ServiceCode := 16#0003, LocalElement := Logix_Status.MemoryRequestData[0], DestinationTag := Logix_Status.MemoryTemp[0], ...)
   MV201_FB : MV_FBD := (Auto := 1, Cmd_Open := 1, AutoInp := 1, ZSO := 1, Open_TM := 15, Close_TM := 15);
   P201_FB : PMP_FBD := (Avl := 1, RunHr := 106.416664, Total_RunHr := 106.416664, Auto := 1, Remote := 1, Start_TM := 3, Stop_TM := 3, Rst := 1, Permissive := -5);
   P202_FB : PMP_FBD := (Avl := 1, RunHr := 0.1, Total_RunHr := 0.1, Auto := 1, Remote := 1, Start_TM := 3, Stop_TM := 3, Rst := 1, Permissive := -5);
   P203_FB : PMP_FBD := (Avl := 1, RunHr := 161.46666, Total_RunHr := 161.46666, Auto := 1, AutoInp := 1, Remote := 1, Start_TM := 3, Stop_TM := 3, Rst := 1, Permissive := -5);
   P204_FB : PMP_FBD := (Avl := 1, RunHr := 0.1, Total_RunHr := 0.1, Auto := 1, Remote := 1, Start_TM := 3, Stop_TM := 3, Rst := 1, Permissive := -5);
   P205_FB : PMP_FBD := (Avl := 1, RunHr := 143.85, Total_RunHr := 143.85, Auto := 1, AutoInp := 1, Remote := 1, Start_TM := 3, Stop_TM := 3, Rst := 1, Permissive := -5);
   P206_FB : PMP_FBD := (Avl := 1, RunHr := 0.06666667, Total_RunHr := 0.06666667, Auto := 1, Remote := 1, Start_TM := 3, Stop_TM := 3, Rst := 1, Permissive := -5);
   P207_FB : PMP_FBD := (Avl := 1, RunHr := 0.016666668, Total_RunHr := 0.016666668, Auto := 1, Remote := 1, Start_TM := 3, Stop_TM := 3, Rst := 1, Permissive := -3);
   P208_FB : PMP_FBD := (Avl := 1, RunHr := 0.016666668, Total_RunHr := 0.016666668, Auto := 1, Remote := 1, Start_TM := 3, Stop_TM := 3, Rst := 1, Permissive := -3);
   P2_P2078_AUTOINP : AUTOINP_UDT;
   P3_LIT301_MSG : MESSAGE;
        MessageParameters(ServiceCode := 16#004c, LocalElement := HMI_LIT301, ...)
   P3_MV301_MSG : MESSAGE;
        MessageParameters(ServiceCode := 16#004c, LocalElement := HMI_MV301, ...)
   P4_AIT402_MSG : MESSAGE;
        MessageParameters(ServiceCode := 16#004c, LocalElement := HMI_AIT402, ...)
   P5_AIT501_PH_MSG : MESSAGE;
        MessageParameters(ServiceCode := 16#004c, LocalElement := HMI_AIT501, ...)
   P5_AIT502_ORP_MSG : MESSAGE;
        MessageParameters(ServiceCode := 16#004c, LocalElement := HMI_AIT502, ...)
   P5_AIT503_COND_MSG : MESSAGE;
        MessageParameters(ServiceCode := 16#004c, LocalElement := HMI_AIT503, ...)
   P5_AIT504_COND_MSG : MESSAGE;
        MessageParameters(ServiceCode := 16#004c, LocalElement := HMI_AIT504, ...)
   P_HCL_DUTY_FB : Duty2_FBD := (AutoInp := 1, Selection := 1, Pmp1_Avl := 1, Pmp2_Avl := 1, Start_Pmp1 := 1);
   P_NACL_DUTY_FB : Duty2_FBD := (Selection := 1, Pmp1_Avl := 1, Pmp2_Avl := 1);
   P_NAOCL_FAC_DUTY_FB : Duty2_FBD := (AutoInp := 1, Selection := 1, Pmp1_Avl := 1, Pmp2_Avl := 1, Start_Pmp1 := 1);
   P_NAOCL_UF_DUTY_FB : Duty2_FBD := (Selection := 2, Pmp1_Avl := 1, Pmp2_Avl := 1);
   P_RAW_WATER_DUTY_FB : Duty2_FBD;
   PLANT_CRITICAL_SD : AUTOINP_UDT;
   REDUNDANT_STATUS : RED_STAT := (Redundancy_status_of_the_controller := 2, Redundancy_state_of_the_partner := 8);
   TEST_REAL : REAL := 2.3664446;
   TON : FBD_TIMER := (TimerEnable := 1, PRE := 1000, ACC := 704, EN := 1, TT := 1);
   TON_FIT102_P1_TM : FBD_TIMER := (PRE := 3000);
   TON_FIT102_P2_TM : FBD_TIMER := (PRE := 3000);
   TON_FIT102_P3_TM : FBD_TIMER := (PRE := 3000);
   TON_FIT102_P4_TM : FBD_TIMER := (PRE := 3000);
   TON_FIT102_P5_TM : FBD_TIMER := (PRE := 3000);
   TON_FIT102_P6_TM : FBD_TIMER := (PRE := 3000);
   TON_FIT102_TM : FBD_TIMER := (TimerEnable := 1, PRE := 3000, ACC := 3002, EN := 1, DN := 1);
   W_AI_AIT_201_COND : INT := 16743;
   W_AI_AIT_201_COND_HTY : BOOL;
   W_AI_AIT_202_PH : INT := 11550;
   W_AI_AIT_202_PH_HTY : BOOL := 1;
   W_AI_AIT_203_ORP : INT := 7064;
   W_AI_AIT_203_ORP_HTY : BOOL := 1;
   W_AI_FIT_201_FLOW : INT := 3263;
   W_AI_FIT_201_FLOW_HTY : BOOL := 1;
END_VAR

PROGRAM MainProgram   (* main routine MainRoutine *)
VAR
   _MIN_P : BOOL;
   _MV_201_SR : DOMINANT_SET := (Out := 1);
   _P_HCL_DUTY_SR : DOMINANT_SET := (Set := 1, Reset := 1, Out := 1);
   _P_NACL_DUTY_SR : DOMINANT_SET := (Reset := 1, OutNot := 1);
   _P_NAOCL_FAC_DUTY_SR : DOMINANT_SET := (Set := 1, Out := 1);
   _P_NAOCL_UF_DUTY_SR : DOMINANT_SET := (Reset := 1, OutNot := 1);
   AIN_FBD_X_01 : AIN_FBD;
   ATTACK : BOOL;
   SEC_TEST : DINT;
END_VAR

ROUTINE Dosing   (* function block diagram *)
   SHEET 1
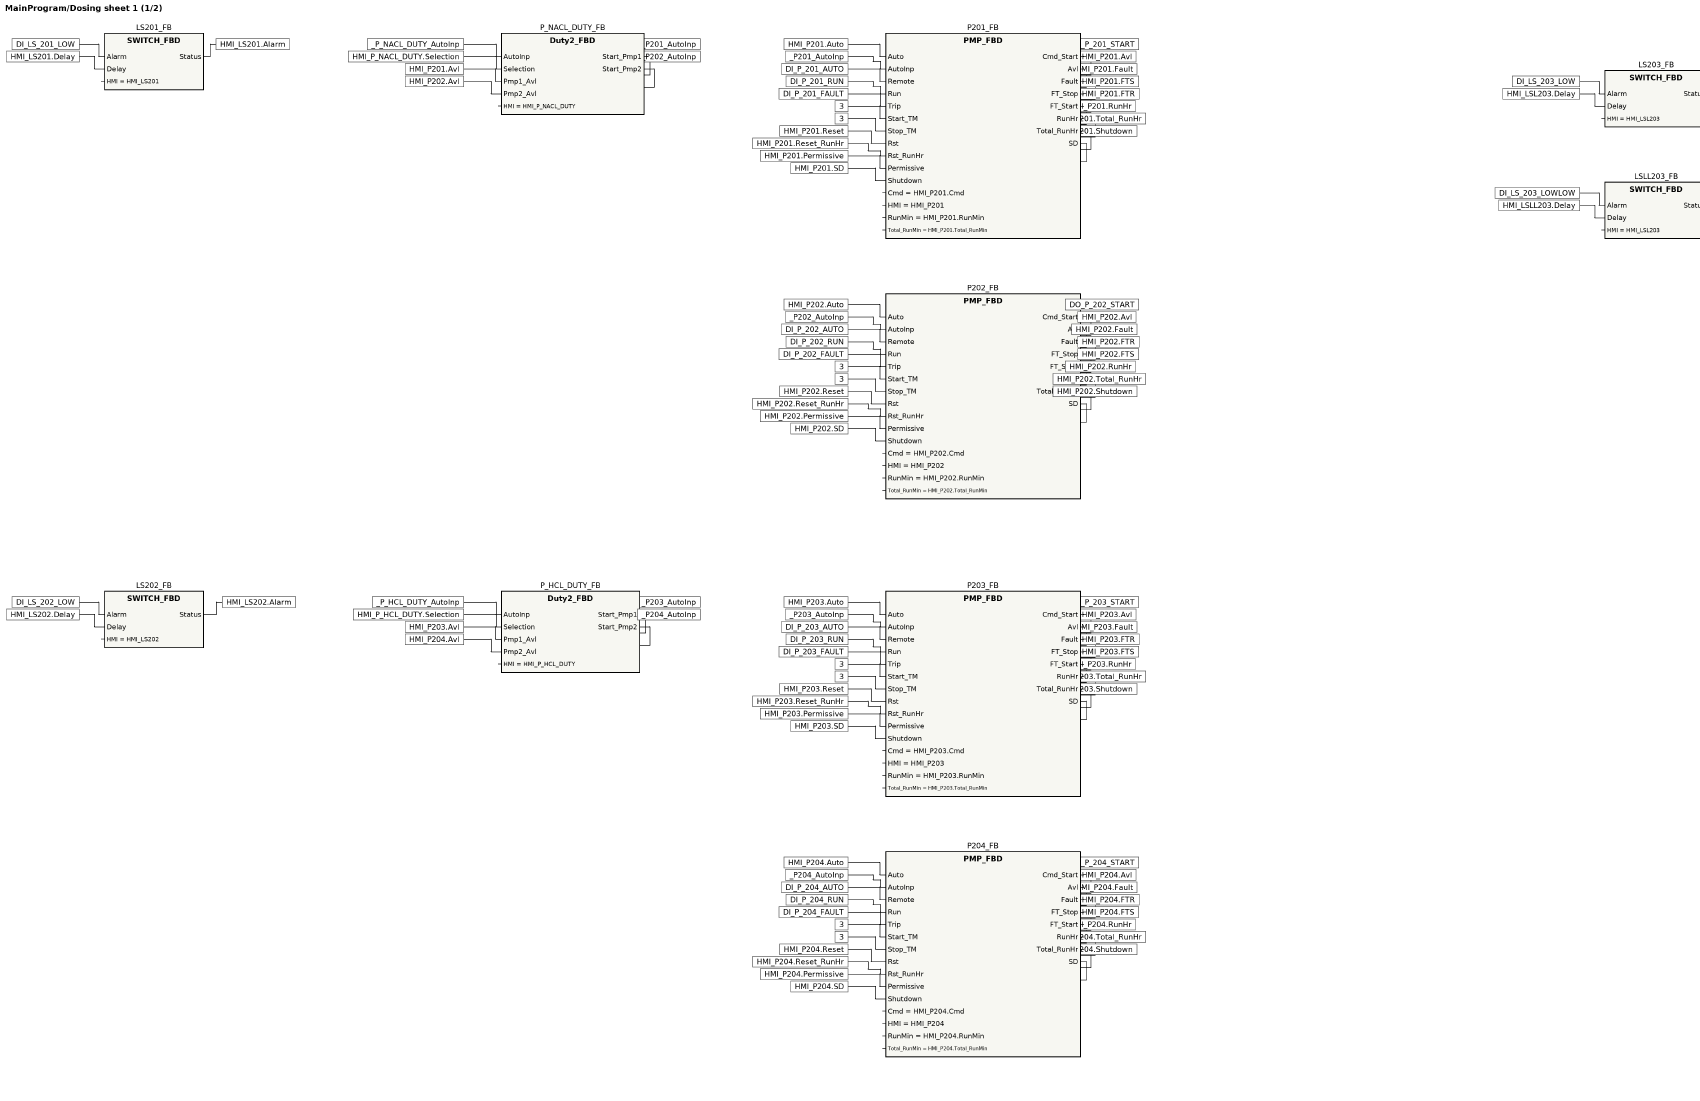
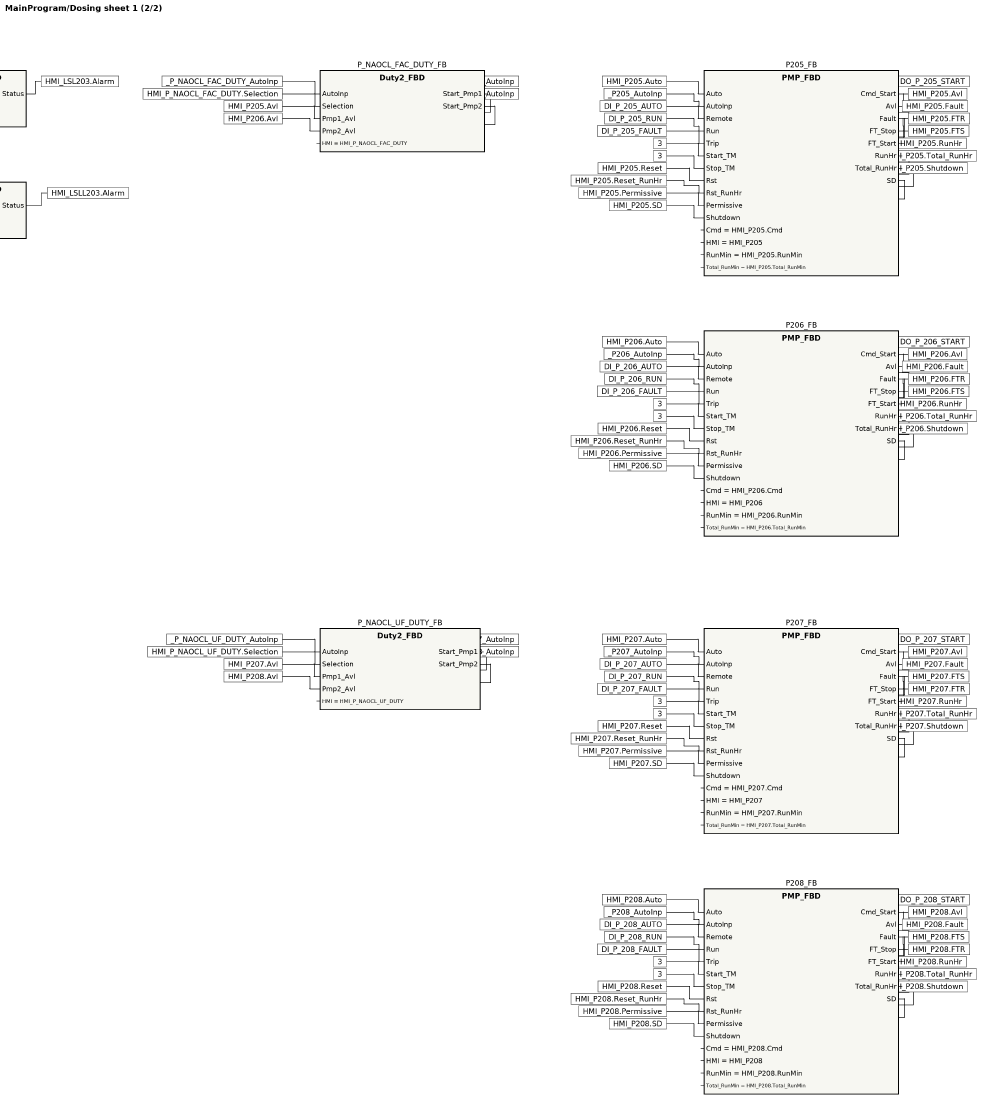
   LS201_FB : SWITCH_FBD(Alarm := DI_LS_201_LOW, Delay := HMI_LS201.Delay, HMI := HMI_LS201);
   LS202_FB : SWITCH_FBD(Alarm := DI_LS_202_LOW, Delay := HMI_LS202.Delay, HMI := HMI_LS202);
   HMI_LS201.Alarm := LS201_FB.Status;
   HMI_LS202.Alarm := LS202_FB.Status;
   P_NACL_DUTY_FB : Duty2_FBD(AutoInp := _P_NACL_DUTY_AutoInp, Selection := HMI_P_NACL_DUTY.Selection, Pmp1_Avl := HMI_P201.Avl, Pmp2_Avl := HMI_P202.Avl, HMI := HMI_P_NACL_DUTY);
   P_HCL_DUTY_FB : Duty2_FBD(AutoInp := _P_HCL_DUTY_AutoInp, Selection := HMI_P_HCL_DUTY.Selection, Pmp1_Avl := HMI_P203.Avl, Pmp2_Avl := HMI_P204.Avl, HMI := HMI_P_HCL_DUTY);
   _P201_AutoInp := P_NACL_DUTY_FB.Start_Pmp1;
   _P202_AutoInp := P_NACL_DUTY_FB.Start_Pmp2;
   _P203_AutoInp := P_HCL_DUTY_FB.Start_Pmp1;
   _P204_AutoInp := P_HCL_DUTY_FB.Start_Pmp2;
   P201_FB : PMP_FBD(Auto := HMI_P201.Auto, AutoInp := _P201_AutoInp, Remote := DI_P_201_AUTO, Run := DI_P_201_RUN, Trip := DI_P_201_FAULT, Start_TM := 3, Stop_TM := 3, Rst := HMI_P201.Reset, Rst_RunHr := HMI_P201.Reset_RunHr, Permissive := HMI_P201.Permissive, Shutdown := HMI_P201.SD, Cmd := HMI_P201.Cmd, HMI := HMI_P201, RunMin := HMI_P201.RunMin, Total_RunMin := HMI_P201.Total_RunMin);
   P202_FB : PMP_FBD(Auto := HMI_P202.Auto, AutoInp := _P202_AutoInp, Remote := DI_P_202_AUTO, Run := DI_P_202_RUN, Trip := DI_P_202_FAULT, Start_TM := 3, Stop_TM := 3, Rst := HMI_P202.Reset, Rst_RunHr := HMI_P202.Reset_RunHr, Permissive := HMI_P202.Permissive, Shutdown := HMI_P202.SD, Cmd := HMI_P202.Cmd, HMI := HMI_P202, RunMin := HMI_P202.RunMin, Total_RunMin := HMI_P202.Total_RunMin);
   P203_FB : PMP_FBD(Auto := HMI_P203.Auto, AutoInp := _P203_AutoInp, Remote := DI_P_203_AUTO, Run := DI_P_203_RUN, Trip := DI_P_203_FAULT, Start_TM := 3, Stop_TM := 3, Rst := HMI_P203.Reset, Rst_RunHr := HMI_P203.Reset_RunHr, Permissive := HMI_P203.Permissive, Shutdown := HMI_P203.SD, Cmd := HMI_P203.Cmd, HMI := HMI_P203, RunMin := HMI_P203.RunMin, Total_RunMin := HMI_P203.Total_RunMin);
   P204_FB : PMP_FBD(Auto := HMI_P204.Auto, AutoInp := _P204_AutoInp, Remote := DI_P_204_AUTO, Run := DI_P_204_RUN, Trip := DI_P_204_FAULT, Start_TM := 3, Stop_TM := 3, Rst := HMI_P204.Reset, Rst_RunHr := HMI_P204.Reset_RunHr, Permissive := HMI_P204.Permissive, Shutdown := HMI_P204.SD, Cmd := HMI_P204.Cmd, HMI := HMI_P204, RunMin := HMI_P204.RunMin, Total_RunMin := HMI_P204.Total_RunMin);
   HMI_P201.Total_RunHr := P201_FB.Total_RunHr;
   HMI_P201.Shutdown := P201_FB.SD;
   HMI_P202.Total_RunHr := P202_FB.Total_RunHr;
   HMI_P202.Shutdown := P202_FB.SD;
   HMI_P203.Total_RunHr := P203_FB.Total_RunHr;
   HMI_P203.Shutdown := P203_FB.SD;
   HMI_P204.Total_RunHr := P204_FB.Total_RunHr;
   HMI_P204.Shutdown := P204_FB.SD;
   DO_P_201_START := P201_FB.Cmd_Start;
   HMI_P201.RunHr := P201_FB.RunHr;
   DO_P_202_START := P202_FB.Cmd_Start;
   HMI_P202.RunHr := P202_FB.RunHr;
   DO_P_203_START := P203_FB.Cmd_Start;
   HMI_P203.RunHr := P203_FB.RunHr;
   DO_P_204_START := P204_FB.Cmd_Start;
   HMI_P204.RunHr := P204_FB.RunHr;
   HMI_P201.Fault := P201_FB.Fault;
   HMI_P202.Fault := P202_FB.Fault;
   HMI_P203.Fault := P203_FB.Fault;
   HMI_P204.Fault := P204_FB.Fault;
   HMI_P201.Avl := P201_FB.Avl;
   HMI_P201.FTS := P201_FB.FT_Stop;
   HMI_P201.FTR := P201_FB.FT_Start;
   HMI_P202.Avl := P202_FB.Avl;
   HMI_P202.FTR := P202_FB.FT_Stop;
   HMI_P202.FTS := P202_FB.FT_Start;
   HMI_P203.Avl := P203_FB.Avl;
   HMI_P203.FTR := P203_FB.FT_Stop;
   HMI_P203.FTS := P203_FB.FT_Start;
   HMI_P204.Avl := P204_FB.Avl;
   HMI_P204.FTR := P204_FB.FT_Stop;
   HMI_P204.FTS := P204_FB.FT_Start;
   LS203_FB : SWITCH_FBD(Alarm := DI_LS_203_LOW, Delay := HMI_LSL203.Delay, HMI := HMI_LSL203);
   LSLL203_FB : SWITCH_FBD(Alarm := DI_LS_203_LOWLOW, Delay := HMI_LSLL203.Delay, HMI := HMI_LSL203);
   HMI_LSL203.Alarm := LS203_FB.Status;
   HMI_LSLL203.Alarm := LSLL203_FB.Status;
   P_NAOCL_FAC_DUTY_FB : Duty2_FBD(AutoInp := _P_NAOCL_FAC_DUTY_AutoInp, Selection := HMI_P_NAOCL_FAC_DUTY.Selection, Pmp1_Avl := HMI_P205.Avl, Pmp2_Avl := HMI_P206.Avl, HMI := HMI_P_NAOCL_FAC_DUTY);
   P_NAOCL_UF_DUTY_FB : Duty2_FBD(AutoInp := _P_NAOCL_UF_DUTY_AutoInp, Selection := HMI_P_NAOCL_UF_DUTY.Selection, Pmp1_Avl := HMI_P207.Avl, Pmp2_Avl := HMI_P208.Avl, HMI := HMI_P_NAOCL_UF_DUTY);
   _P205_AutoInp := P_NAOCL_FAC_DUTY_FB.Start_Pmp1;
   _P206_AutoInp := P_NAOCL_FAC_DUTY_FB.Start_Pmp2;
   _P207_AutoInp := P_NAOCL_UF_DUTY_FB.Start_Pmp1;
   _P208_AutoInp := P_NAOCL_UF_DUTY_FB.Start_Pmp2;
   P205_FB : PMP_FBD(Auto := HMI_P205.Auto, AutoInp := _P205_AutoInp, Remote := DI_P_205_AUTO, Run := DI_P_205_RUN, Trip := DI_P_205_FAULT, Start_TM := 3, Stop_TM := 3, Rst := HMI_P205.Reset, Rst_RunHr := HMI_P205.Reset_RunHr, Permissive := HMI_P205.Permissive, Shutdown := HMI_P205.SD, Cmd := HMI_P205.Cmd, HMI := HMI_P205, RunMin := HMI_P205.RunMin, Total_RunMin := HMI_P205.Total_RunMin);
   P206_FB : PMP_FBD(Auto := HMI_P206.Auto, AutoInp := _P206_AutoInp, Remote := DI_P_206_AUTO, Run := DI_P_206_RUN, Trip := DI_P_206_FAULT, Start_TM := 3, Stop_TM := 3, Rst := HMI_P206.Reset, Rst_RunHr := HMI_P206.Reset_RunHr, Permissive := HMI_P206.Permissive, Shutdown := HMI_P206.SD, Cmd := HMI_P206.Cmd, HMI := HMI_P206, RunMin := HMI_P206.RunMin, Total_RunMin := HMI_P206.Total_RunMin);
   P207_FB : PMP_FBD(Auto := HMI_P207.Auto, AutoInp := _P207_AutoInp, Remote := DI_P_207_AUTO, Run := DI_P_207_RUN, Trip := DI_P_207_FAULT, Start_TM := 3, Stop_TM := 3, Rst := HMI_P207.Reset, Rst_RunHr := HMI_P207.Reset_RunHr, Permissive := HMI_P207.Permissive, Shutdown := HMI_P207.SD, Cmd := HMI_P207.Cmd, HMI := HMI_P207, RunMin := HMI_P207.RunMin, Total_RunMin := HMI_P207.Total_RunMin);
   P208_FB : PMP_FBD(Auto := HMI_P208.Auto, AutoInp := _P208_AutoInp, Remote := DI_P_208_AUTO, Run := DI_P_208_RUN, Trip := DI_P_208_FAULT, Start_TM := 3, Stop_TM := 3, Rst := HMI_P208.Reset, Rst_RunHr := HMI_P208.Reset_RunHr, Permissive := HMI_P208.Permissive, Shutdown := HMI_P208.SD, Cmd := HMI_P208.Cmd, HMI := HMI_P208, RunMin := HMI_P208.RunMin, Total_RunMin := HMI_P208.Total_RunMin);
   HMI_P205.Total_RunHr := P205_FB.Total_RunHr;
   HMI_P205.Shutdown := P205_FB.SD;
   HMI_P206.Total_RunHr := P206_FB.Total_RunHr;
   HMI_P206.Shutdown := P206_FB.SD;
   HMI_P207.Total_RunHr := P207_FB.Total_RunHr;
   HMI_P207.Shutdown := P207_FB.SD;
   HMI_P208.Total_RunHr := P208_FB.Total_RunHr;
   HMI_P208.Shutdown := P208_FB.SD;
   DO_P_205_START := P205_FB.Cmd_Start;
   HMI_P205.RunHr := P205_FB.RunHr;
   DO_P_206_START := P206_FB.Cmd_Start;
   HMI_P206.RunHr := P206_FB.RunHr;
   DO_P_207_START := P207_FB.Cmd_Start;
   HMI_P207.RunHr := P207_FB.RunHr;
   DO_P_208_START := P208_FB.Cmd_Start;
   HMI_P208.RunHr := P208_FB.RunHr;
   HMI_P205.Fault := P205_FB.Fault;
   HMI_P206.Fault := P206_FB.Fault;
   HMI_P207.Fault := P207_FB.Fault;
   HMI_P208.Fault := P208_FB.Fault;
   HMI_P205.Avl := P205_FB.Avl;
   HMI_P205.FTR := P205_FB.FT_Stop;
   HMI_P205.FTS := P205_FB.FT_Start;
   HMI_P206.Avl := P206_FB.Avl;
   HMI_P206.FTR := P206_FB.FT_Stop;
   HMI_P206.FTS := P206_FB.FT_Start;
   HMI_P207.Avl := P207_FB.Avl;
   HMI_P207.FTS := P207_FB.FT_Stop;
   HMI_P207.FTR := P207_FB.FT_Start;
   HMI_P208.Avl := P208_FB.Avl;
   HMI_P208.FTS := P208_FB.FT_Stop;
   HMI_P208.FTR := P208_FB.FT_Start;
END_ROUTINE

ROUTINE IO   (* structured text *)
   (*DIGITAL INPUTS*)
   DI_WIFI_PLC_2	:=RIO2:0:I.Data.0;
   DI_WIFI_RIO_2	:=RIO2:0:I.Data.1;
   DI_P_201_AUTO	:=RIO2:0:I.Data.2;
   DI_P_201_RUN	:=RIO2:0:I.Data.3;
   DI_P_201_FAULT	:=RIO2:0:I.Data.4;
   DI_P_202_AUTO	:=RIO2:0:I.Data.5;
   DI_P_202_RUN	:=RIO2:0:I.Data.6;
   DI_P_202_FAULT	:=RIO2:0:I.Data.7;
   DI_P_203_AUTO	:=RIO2:0:I.Data.8;
   DI_P_203_RUN	:=RIO2:0:I.Data.9;
   DI_P_203_FAULT	:=RIO2:0:I.Data.10;
   DI_P_204_AUTO	:=RIO2:0:I.Data.11;
   DI_P_204_RUN	:=RIO2:0:I.Data.12;
   DI_P_204_FAULT	:=RIO2:0:I.Data.13;
   DI_P_205_AUTO	:=RIO2:0:I.Data.14;
   DI_P_205_RUN	:=RIO2:0:I.Data.15;
   DI_P_205_FAULT	:=RIO2:0:I.Data.16;
   DI_P_206_AUTO	:=RIO2:0:I.Data.17;
   DI_P_206_RUN	:=RIO2:0:I.Data.18;
   DI_P_206_FAULT	:=RIO2:0:I.Data.19;
   DI_P_207_AUTO	:=RIO2:0:I.Data.20;
   DI_P_207_RUN	:=RIO2:0:I.Data.21;
   DI_P_207_FAULT	:=RIO2:0:I.Data.22;
   DI_P_208_AUTO	:=RIO2:0:I.Data.23;
   DI_P_208_RUN	:=RIO2:0:I.Data.24;
   DI_P_208_FAULT	:=RIO2:0:I.Data.25;
   DI_MV_201_ZSO	:=RIO2:0:I.Data.26;
   DI_MV_201_ZSC	:=RIO2:0:I.Data.27;
   DI_LS_201_LOW	:=RIO2:0:I.Data.28;
   DI_LS_202_LOW	:=RIO2:0:I.Data.29;
   DI_LS_203_LOW	:=RIO2:0:I.Data.30;
   DI_LS_203_LOWLOW:=RIO2:0:I.Data.31;
   
   (*DIGITAL OUTPUTS*)
   RIO2:1:O.0	:=DO_P_201_START;
   RIO2:1:O.1	:=DO_P_202_START;
   RIO2:1:O.2	:=DO_P_203_START;
   RIO2:1:O.3	:=DO_P_204_START;
   RIO2:1:O.4	:=DO_P_205_START;
   RIO2:1:O.5	:=DO_P_206_START;
   RIO2:1:O.6	:=DO_P_207_START;
   RIO2:1:O.7	:=DO_P_208_START;
   RIO2:1:O.8	:=DO_MV_201_OPEN;
   RIO2:1:O.9	:=DO_MV_201_CLOSE;
   RIO2:1:O.10	:=DO_RIO2_SPARE_10;
   RIO2:1:O.11	:=DO_RIO2_SPARE_11;
   
   (*ANALOG INPUTS*)
   AI_FIT_201_FLOW	:=RIO2:2:I.Ch0Data;
   AI_AIT_201_COND	:=RIO2:2:I.Ch1Data;
   AI_AIT_202_PH	:=RIO2:2:I.Ch2Data;
   AI_AIT_203_ORP	:=RIO2:2:I.Ch3Data;
   AI_RIO2_SPARE_04:=RIO2:2:I.Ch4Data;
   AI_RIO2_SPARE_05:=RIO2:2:I.Ch5Data;
   AI_RIO2_SPARE_06:=RIO2:2:I.Ch6Data;
   AI_RIO2_SPARE_07:=RIO2:2:I.Ch7Data;
   AI_RIO2_SPARE_08:=RIO2:2:I.Ch8Data;
   AI_RIO2_SPARE_09:=RIO2:2:I.Ch9Data;
   AI_RIO2_SPARE_10:=RIO2:2:I.Ch10Data;
   AI_RIO2_SPARE_11:=RIO2:2:I.Ch11Data;
   
   AI_FIT_201_FLOW_HTY		:=(NOT RIO2:2:I.GeneralFault);
   AI_AIT_201_COND_HTY		:=(NOT RIO2:2:I.GeneralFault);
   AI_AIT_202_PH_HTY		:=(NOT RIO2:2:I.GeneralFault);
   AI_AIT_203_ORP_HTY		:=(NOT RIO2:2:I.GeneralFault);
   AI_RIO2_SPARE_04_HTY	:=(NOT RIO2:2:I.GeneralFault);
   AI_RIO2_SPARE_05_HTY	:=(NOT RIO2:2:I.GeneralFault);
   AI_RIO2_SPARE_06_HTY	:=(NOT RIO2:2:I.GeneralFault);
   AI_RIO2_SPARE_07_HTY	:=(NOT RIO2:2:I.GeneralFault);
   AI_RIO2_SPARE_08_HTY	:=(NOT RIO2:2:I.GeneralFault);
   AI_RIO2_SPARE_09_HTY	:=(NOT RIO2:2:I.GeneralFault);
   AI_RIO2_SPARE_10_HTY	:=(NOT RIO2:2:I.GeneralFault);
   AI_RIO2_SPARE_11_HTY	:=(NOT RIO2:2:I.GeneralFault);
   
   (*WIRELESS ANALOG INPUTS*)
   W_AI_FIT_201_FLOW	:=WRIO2:1:I.Ch0Data;
   W_AI_AIT_201_COND	:=WRIO2:1:I.Ch1Data;
   W_AI_AIT_202_PH		:=WRIO2:1:I.Ch2Data;
   W_AI_AIT_203_ORP	:=WRIO2:1:I.Ch3Data;
   
   W_AI_FIT_201_FLOW_HTY	:=(NOT WRIO2:1:I.Ch0Fault);
   W_AI_AIT_201_COND_HTY	:=(NOT WRIO2:1:I.Ch1Fault);
   W_AI_AIT_202_PH_HTY		:=(NOT WRIO2:1:I.Ch2Fault);
   W_AI_AIT_203_ORP_HTY	:=(NOT WRIO2:1:I.Ch3Fault);
   
   (*Wireless Selction*)
   HMI_WIFI.PLC_WIFI		:= DI_WIFI_PLC_2;
   HMI_WIFI.RIO_WIFI		:= DI_WIFI_RIO_2;
   
END_ROUTINE

ROUTINE Logix_Status   (* ladder *)
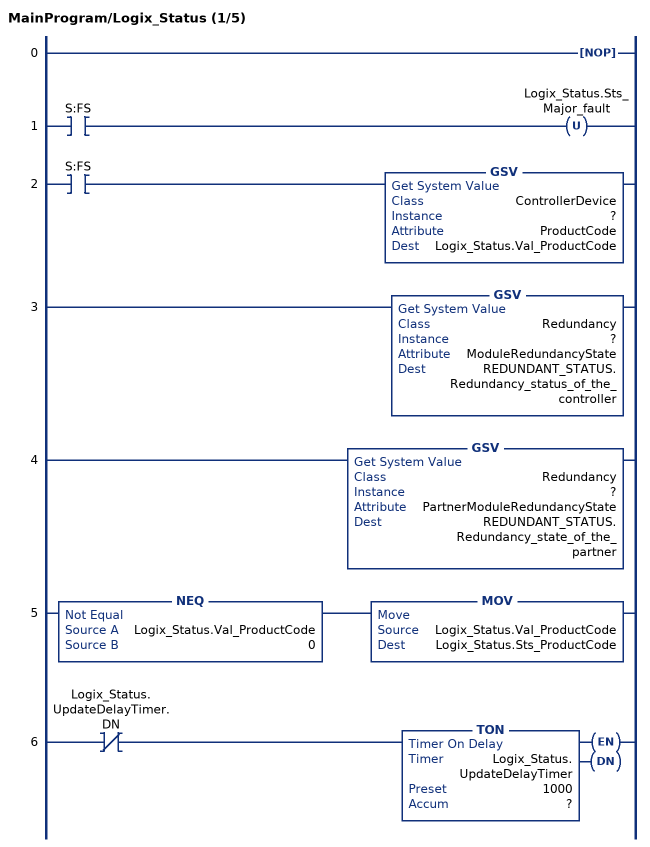
   0: NOP();
   1: XIC(S:FS)OTU(Logix_Status.Sts_Major_fault);
   2: XIC(S:FS)GSV(ControllerDevice,?,ProductCode,Logix_Status.Val_ProductCode);
   3: GSV(Redundancy,?,ModuleRedundancyState,REDUNDANT_STATUS.Redundancy_status_of_the_controller);
   4: GSV(Redundancy,?,PartnerModuleRedundancyState,REDUNDANT_STATUS.Redundancy_state_of_the_partner);
   5: NEQ(Logix_Status.Val_ProductCode,0)MOV(Logix_Status.Val_ProductCode,Logix_Status.Sts_ProductCode);
   6: XIO(Logix_Status.UpdateDelayTimer.DN)TON(Logix_Status.UpdateDelayTimer,?,?);
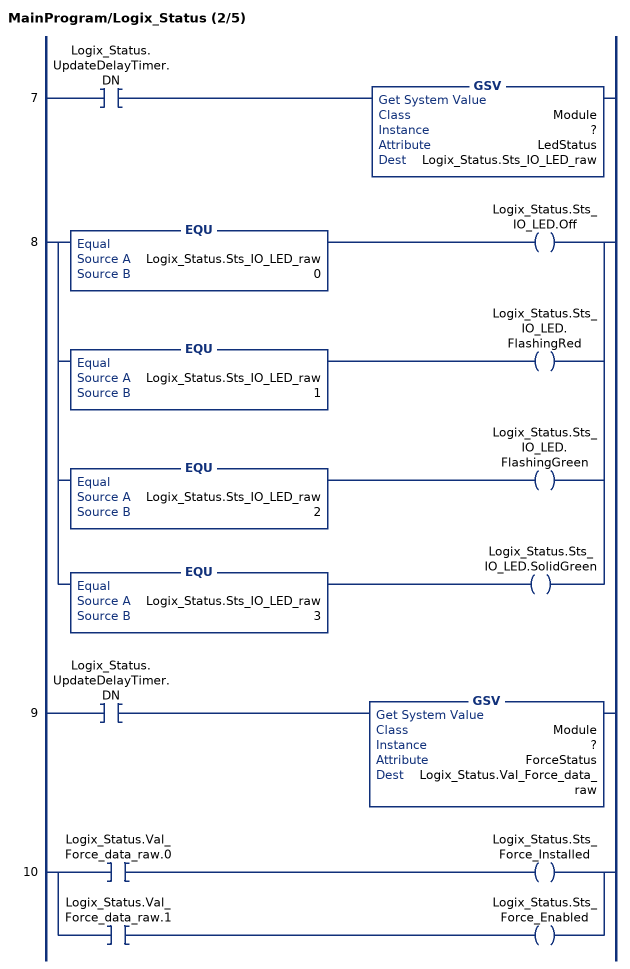
   7: XIC(Logix_Status.UpdateDelayTimer.DN)GSV(Module,?,LedStatus,Logix_Status.Sts_IO_LED_raw);
   8: [EQU(Logix_Status.Sts_IO_LED_raw,0) OTE(Logix_Status.Sts_IO_LED.Off) ,EQU(Logix_Status.Sts_IO_LED_raw,1) OTE(Logix_Status.Sts_IO_LED.FlashingRed) ,EQU(Logix_Status.Sts_IO_LED_raw,2) OTE(Logix_Status.Sts_IO_LED.FlashingGreen) ,EQU(Logix_Status.Sts_IO_LED_raw,3) OTE(Logix_Status.Sts_IO_LED.SolidGreen) ];
   9: XIC(Logix_Status.UpdateDelayTimer.DN)GSV(Module,?,ForceStatus,Logix_Status.Val_Force_data_raw);
   10: [XIC(Logix_Status.Val_Force_data_raw.0) OTE(Logix_Status.Sts_Force_Installed) ,XIC(Logix_Status.Val_Force_data_raw.1) OTE(Logix_Status.Sts_Force_Enabled) ];
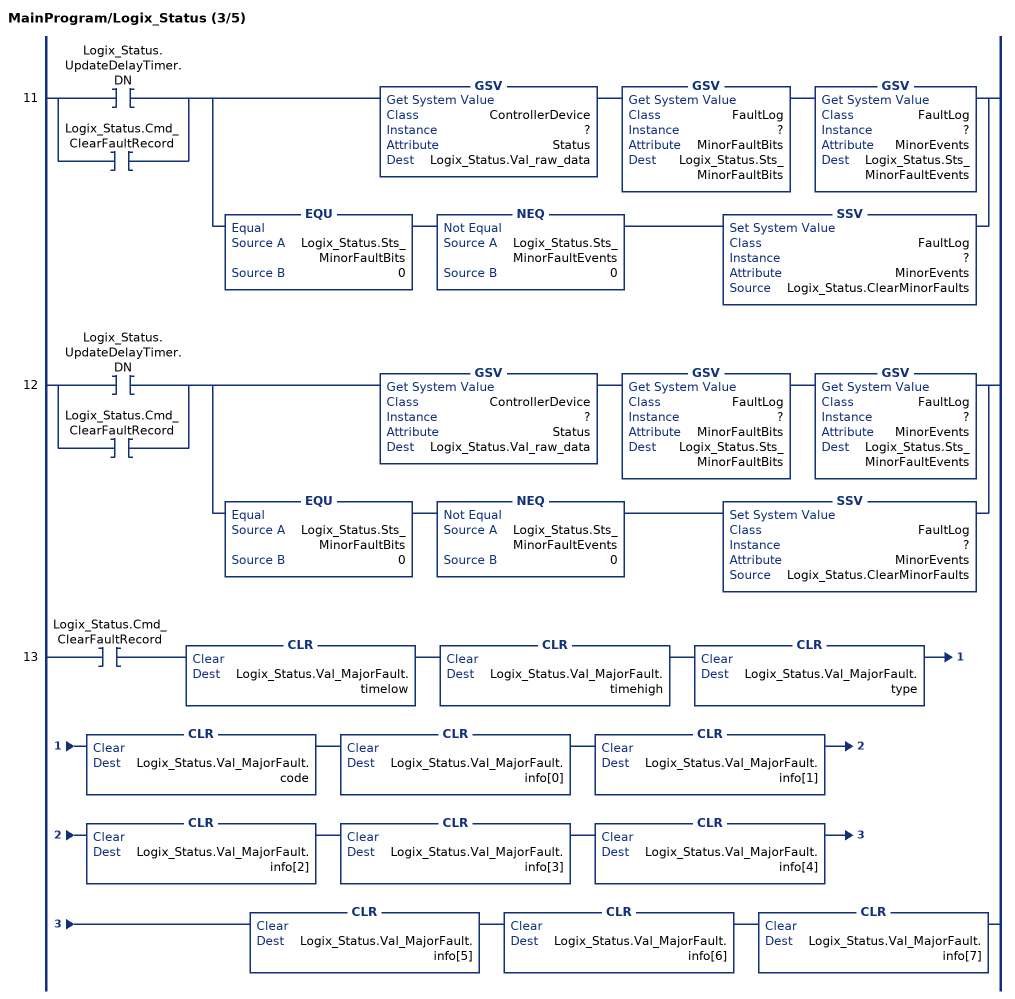
   11: [XIC(Logix_Status.UpdateDelayTimer.DN) ,XIC(Logix_Status.Cmd_ClearFaultRecord) ][GSV(ControllerDevice,?,Status,Logix_Status.Val_raw_data) GSV(FaultLog,?,MinorFaultBits,Logix_Status.Sts_MinorFaultBits) GSV(FaultLog,?,MinorEvents,Logix_Status.Sts_MinorFaultEvents) ,EQU(Logix_Status.Sts_MinorFaultBits,0) NEQ(Logix_Status.Sts_MinorFaultEvents,0) SSV(FaultLog,?,MinorEvents,Logix_Status.ClearMinorFaults) ];
   12: [XIC(Logix_Status.UpdateDelayTimer.DN) ,XIC(Logix_Status.Cmd_ClearFaultRecord) ][GSV(ControllerDevice,?,Status,Logix_Status.Val_raw_data) GSV(FaultLog,?,MinorFaultBits,Logix_Status.Sts_MinorFaultBits) GSV(FaultLog,?,MinorEvents,Logix_Status.Sts_MinorFaultEvents) ,EQU(Logix_Status.Sts_MinorFaultBits,0) NEQ(Logix_Status.Sts_MinorFaultEvents,0) SSV(FaultLog,?,MinorEvents,Logix_Status.ClearMinorFaults) ];
   13: XIC(Logix_Status.Cmd_ClearFaultRecord)CLR(Logix_Status.Val_MajorFault.timelow)CLR(Logix_Status.Val_MajorFault.timehigh)CLR(Logix_Status.Val_MajorFault.type)CLR(Logix_Status.Val_MajorFault.code)CLR(Logix_Status.Val_MajorFault.info[0])CLR(Logix_Status.Val_MajorFault.info[1])CLR(Logix_Status.Val_MajorFault.info[2])CLR(Logix_Status.Val_MajorFault.info[3])CLR(Logix_Status.Val_MajorFault.info[4])CLR(Logix_Status.Val_MajorFault.info[5])CLR(Logix_Status.Val_MajorFault.info[6])CLR(Logix_Status.Val_MajorFault.info[7]);
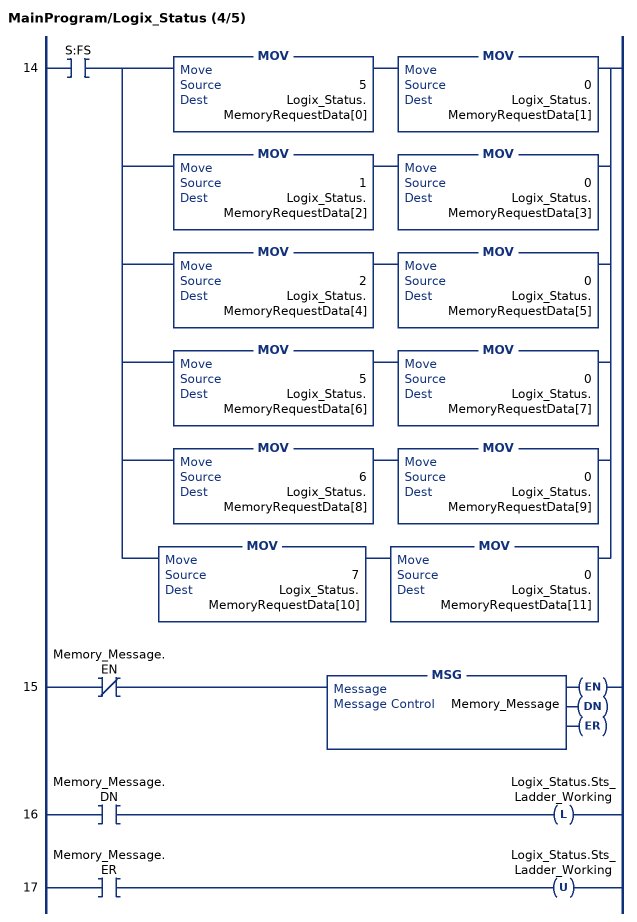
   14: XIC(S:FS)[MOV(5,Logix_Status.MemoryRequestData[0]) MOV(0,Logix_Status.MemoryRequestData[1]) ,MOV(1,Logix_Status.MemoryRequestData[2]) MOV(0,Logix_Status.MemoryRequestData[3]) ,MOV(2,Logix_Status.MemoryRequestData[4]) MOV(0,Logix_Status.MemoryRequestData[5]) ,MOV(5,Logix_Status.MemoryRequestData[6]) MOV(0,Logix_Status.MemoryRequestData[7]) ,MOV(6,Logix_Status.MemoryRequestData[8]) MOV(0,Logix_Status.MemoryRequestData[9]) ,MOV(7,Logix_Status.MemoryRequestData[10]) MOV(0,Logix_Status.MemoryRequestData[11]) ];
   15: XIO(Memory_Message.EN)MSG(Memory_Message);
   16: XIC(Memory_Message.DN)OTL(Logix_Status.Sts_Ladder_Working);
   17: XIC(Memory_Message.ER)OTU(Logix_Status.Sts_Ladder_Working);
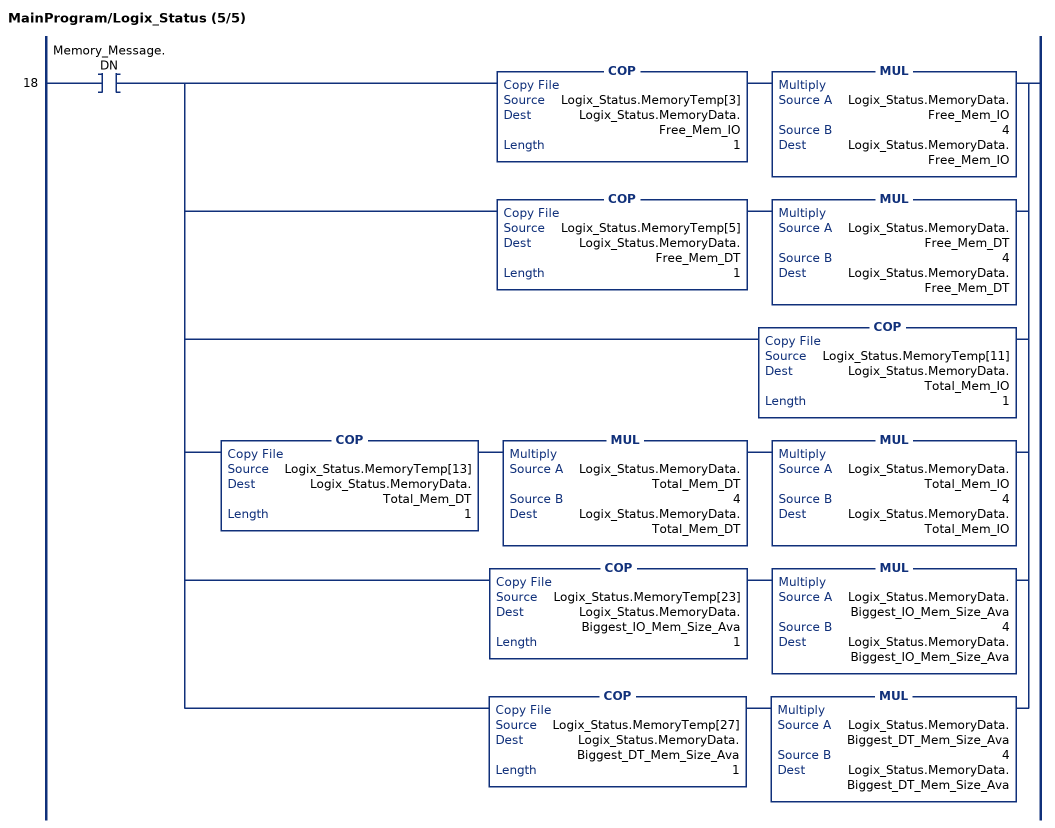
   18: XIC(Memory_Message.DN)[COP(Logix_Status.MemoryTemp[3],Logix_Status.MemoryData.Free_Mem_IO,1) MUL(Logix_Status.MemoryData.Free_Mem_IO,4,Logix_Status.MemoryData.Free_Mem_IO) ,COP(Logix_Status.MemoryTemp[5],Logix_Status.MemoryData.Free_Mem_DT,1) MUL(Logix_Status.MemoryData.Free_Mem_DT,4,Logix_Status.MemoryData.Free_Mem_DT) ,COP(Logix_Status.MemoryTemp[11],Logix_Status.MemoryData.Total_Mem_IO,1) ,COP(Logix_Status.MemoryTemp[13],Logix_Status.MemoryData.Total_Mem_DT,1) MUL(Logix_Status.MemoryData.Total_Mem_DT,4,Logix_Status.MemoryData.Total_Mem_DT) MUL(Logix_Status.MemoryData.Total_Mem_IO,4,Logix_Status.MemoryData.Total_Mem_IO) ,COP(Logix_Status.MemoryTemp[23],Logix_Status.MemoryData.Biggest_IO_Mem_Size_Ava,1) MUL(Logix_Status.MemoryData.Biggest_IO_Mem_Size_Ava,4,Logix_Status.MemoryData.Biggest_IO_Mem_Size_Ava) ,COP(Logix_Status.MemoryTemp[27],Logix_Status.MemoryData.Biggest_DT_Mem_Size_Ava,1) MUL(Logix_Status.MemoryData.Biggest_DT_Mem_Size_Ava,4,Logix_Status.MemoryData.Biggest_DT_Mem_Size_Ava) ];
END_ROUTINE

ROUTINE Main_Seq   (* structured text *)
   
   
   
   
   (*
   IF HMI_PLANT.STOP THEN
   	HMI_P2_STATE:=1;
   END_IF;
   *)
   
   (*
   IF HMI_PLANT.STOP THEN
   	HMI_P2_SHUTDOWN:=1;
   END_IF;
   *)
   
   IF HMI_PLANT.STOP OR PLANT_CRITICAL_SD.ON THEN
   	HMI_P2_SHUTDOWN:=1;
   END_IF;
   
   
   (*
   if S:FS then
   	HMI_P2_STATE := 1;
   end_if;
   *)
   
   
   
   (*-----------WRITE FAULT CONDITION--------------*)
   
   CASE HMI_P2_STATE OF
   	1:(*PLANT IN STANDBY*)
   		_MV201_AutoInp				:=0;
   		_P_NACL_DUTY_AutoInp		:=0;
   		_P_HCL_DUTY_AutoInp			:=0;
   		_P_NAOCL_FAC_DUTY_AutoInp	:=0;
   		_P_NAOCL_UF_DUTY_AutoInp	:=0;
   
   		IF HMI_P2_PERMISSIVE.ON AND HMI_PLANT.START THEN
   			HMI_P2_STATE:=2;
   		END_IF;
   
   	2:(*OPEN RAW WATER OUTLET VALVE, MV201*)
   		(*MV-201 , Raw Water Outlet Valve Control*)
   		_MV_201_SR.EnableIn		:=1;
   		_MV_201_SR.Set			:=HMI_LIT301.AL;
   		_MV_201_SR.Reset		:=HMI_LIT301.AH;
   		SETD(_MV_201_SR);
   		_MV201_AutoInp			:= _MV_201_SR.Out;
   
   		(*P-201/2 , Cond NACL Dosing Pump Control*)
   		_P_NACL_DUTY_SR.EnableIn	:= 1;
   		_P_NACL_DUTY_SR.Set			:= HMI_MV201.Status=2 AND (HMI_AIT201.AL) AND (NOT HMI_AIT503.AH) ;
   		_P_NACL_DUTY_SR.Reset		:= HMI_MV201.Status<>2 OR (HMI_AIT201.AH) OR (HMI_AIT503.AH) OR  HMI_LS201.Alarm OR HMI_FIT201.ALL  ;
   		SETD(_P_NACL_DUTY_SR);
   		_P_NACL_DUTY_AutoInp		:= _P_NACL_DUTY_SR.Out;
   
   		(*P-203/4 , PH HCL Dosing Pump Control*)
   		_P_HCL_DUTY_SR.EnableIn		:= 1;
   		_P_HCL_DUTY_SR.Set			:= HMI_MV201.Status=2 AND (HMI_AIT202.AH) ;
   		_P_HCL_DUTY_SR.Reset		:= HMI_MV201.Status<>2 OR (HMI_AIT202.AL) OR  HMI_LS202.Alarm OR HMI_FIT201.ALL ;
   		SETD(_P_HCL_DUTY_SR);
   		_P_HCL_DUTY_AutoInp			:= _P_HCL_DUTY_SR.Out;
   
   		(*P-205/6 ,ORP NAOCL FAC Dosing Pump Control*)
   		_P_NAOCL_FAC_DUTY_SR.EnableIn		:= 1;
   		_P_NAOCL_FAC_DUTY_SR.Set			:= HMI_MV201.Status=2 AND (HMI_AIT203.AL) AND (NOT HMI_AIT402.AH) ;
   		_P_NAOCL_FAC_DUTY_SR.Reset			:= HMI_MV201.Status<>2 OR (HMI_AIT203.AH) OR (HMI_AIT402.AH) OR HMI_LSL203.Alarm ;
   		SETD(_P_NAOCL_FAC_DUTY_SR);
   		_P_NAOCL_FAC_DUTY_AutoInp			:= _P_NAOCL_FAC_DUTY_SR.Out;
   
   		(*P-207/8 ,ORP NAOCL UF Dosing Pump Control*)
   		_P_NAOCL_UF_DUTY_SR.EnableIn		:= 1;
   		_P_NAOCL_UF_DUTY_SR.Set				:= P2_P2078_AUTOINP.ON;
   		_P_NAOCL_UF_DUTY_SR.Reset			:= NOT P2_P2078_AUTOINP.ON;
   		SETD(_P_NAOCL_UF_DUTY_SR);
   		_P_NAOCL_UF_DUTY_AutoInp			:= _P_NAOCL_UF_DUTY_SR.Out;
   
   		HMI_P2_READY	:=1;
   
   		IF HMI_P2_SHUTDOWN THEN
   			IF HMI_LIT301.AH THEN
   				HMI_P2_STATE	:=1;
   				HMI_P2_SHUTDOWN	:=0;
   			END_IF;
   
   
   		END_IF;
   
   
   
   ELSE
   	HMI_P2_STATE:=1;
   END_CASE;
   
   
   
   
   
   
   
   
   
   
   
   
   
   
   
   
   
   
   
   
   
   
   
   
   
   
END_ROUTINE

ROUTINE MainRoutine   (* ladder *)
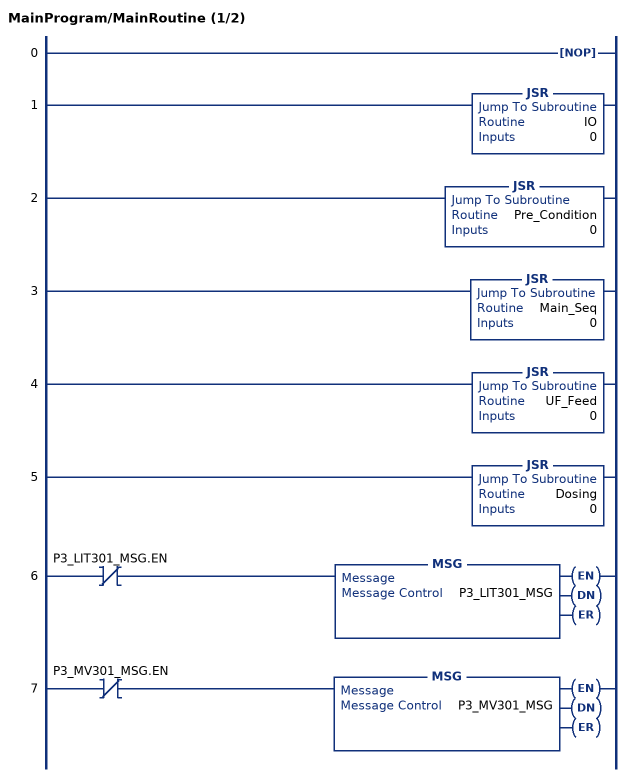
   0: NOP();
   1: JSR(IO,0);
   2: JSR(Pre_Condition,0);
   3: JSR(Main_Seq,0);
   4: JSR(UF_Feed,0);
   5: JSR(Dosing,0);
   6: XIO(P3_LIT301_MSG.EN)MSG(P3_LIT301_MSG);
   7: XIO(P3_MV301_MSG.EN)MSG(P3_MV301_MSG);
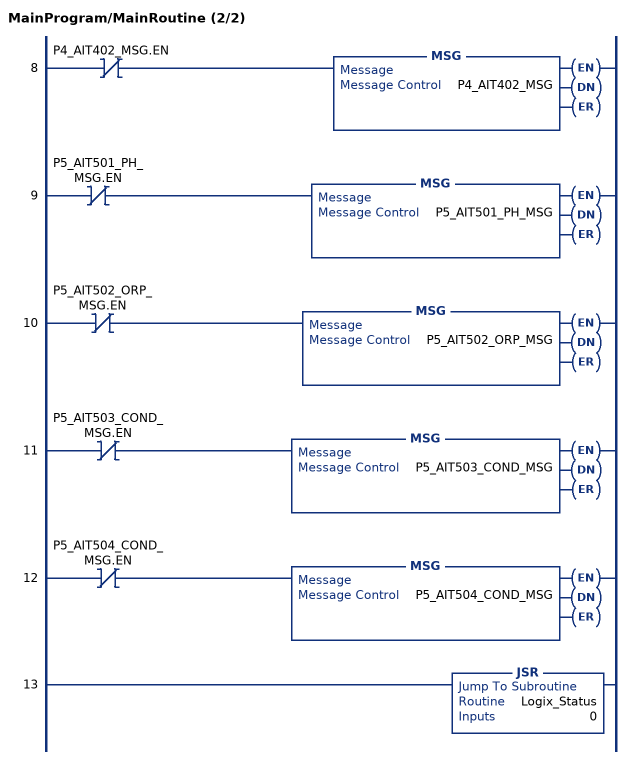
   8: XIO(P4_AIT402_MSG.EN)MSG(P4_AIT402_MSG);
   9: XIO(P5_AIT501_PH_MSG.EN)MSG(P5_AIT501_PH_MSG);
   10: XIO(P5_AIT502_ORP_MSG.EN)MSG(P5_AIT502_ORP_MSG);
   11: XIO(P5_AIT503_COND_MSG.EN)MSG(P5_AIT503_COND_MSG);
   12: XIO(P5_AIT504_COND_MSG.EN)MSG(P5_AIT504_COND_MSG);
   13: JSR(Logix_Status,0);
END_ROUTINE

ROUTINE Pre_Condition   (* structured text *)
   (*RESET ALL INSTRUMENT*)
   IF HMI_PLANT_RESET.ON THEN
   	HMI_MV201.Reset	:=1;
   	HMI_P201.Reset 	:=1;
   	HMI_P202.Reset	:=1;
   	HMI_P203.Reset 	:=1;
   	HMI_P204.Reset	:=1;
   	HMI_P205.Reset	:=1;
   	HMI_P206.Reset	:=1;
   	HMI_P207.Reset 	:=1;
   	HMI_P208.Reset	:=1;
   END_IF;
   
   (*ALL INSTRUMENT IN AUTO MODE*)
   IF HMI_PLANT_AUTO.ON THEN
   	HMI_MV201.Auto	:=1;
   	HMI_P201.Auto 	:=1;
   	HMI_P202.Auto	:=1;
   	HMI_P203.Auto 	:=1;
   	HMI_P204.Auto	:=1;
   	HMI_P205.Auto	:=1;
   	HMI_P206.Auto	:=1;
   	HMI_P207.Auto 	:=1;
   	HMI_P208.Auto	:=1;
   END_IF;
   
   (*ALL INSTRUMENT IN MANUAL MODE*)
   IF HMI_PLANT_AUTO.OFF THEN
   	HMI_MV201.Auto	:=0;
   	HMI_P201.Auto 	:=0;
   	HMI_P202.Auto	:=0;
   	HMI_P203.Auto 	:=0;
   	HMI_P204.Auto	:=0;
   	HMI_P205.Auto	:=0;
   	HMI_P206.Auto	:=0;
   	HMI_P207.Auto 	:=0;
   	HMI_P208.Auto	:=0;
   END_IF;
   
   (*P2 PERMISSIVE*)
   HMI_P2_PERMISSIVE.ON 	:= HMI_MV201.Avl
   						AND (HMI_P201.Avl OR HMI_P202.Avl)
   						AND (HMI_P203.Avl OR HMI_P204.Avl)
   						AND (HMI_P205.Avl OR HMI_P206.Avl);
   						(*AND (HMI_P207.Avl OR HMI_P208.Avl);*)
   
   (*Enable Flow Totalising*)
   _FIT201_Tot_Enb 		:= HMI_MV201.status=2;
   
   TON_FIT102_P1_TM.PRE 			:= 	3*1000;
   TON_FIT102_P1_TM.TimerEnable 	:=  HMI_FIT201.ALL AND HMI_MV201.STATUS=2 AND HMI_P201.STATUS=2;
   TONR(TON_FIT102_P1_TM);
   
   TON_FIT102_P2_TM.PRE 			:= 	3*1000;
   TON_FIT102_P2_TM.TimerEnable 	:=  HMI_FIT201.ALL AND HMI_MV201.STATUS=2 AND HMI_P202.STATUS=2;
   TONR(TON_FIT102_P2_TM);
   
   TON_FIT102_P3_TM.PRE 			:= 	3*1000;
   TON_FIT102_P3_TM.TimerEnable 	:=  HMI_FIT201.ALL AND HMI_MV201.STATUS=2 AND HMI_P203.STATUS=2;
   TONR(TON_FIT102_P3_TM);
   
   TON_FIT102_P4_TM.PRE 			:= 	3*1000;
   TON_FIT102_P4_TM.TimerEnable 	:=  HMI_FIT201.ALL AND HMI_MV201.STATUS=2 AND HMI_P204.STATUS=2;
   TONR(TON_FIT102_P4_TM);
   
   TON_FIT102_P5_TM.PRE 			:= 	3*1000;
   TON_FIT102_P5_TM.TimerEnable 	:=  HMI_FIT201.ALL AND HMI_MV201.STATUS=2 AND HMI_P205.STATUS=2;
   TONR(TON_FIT102_P5_TM);
   
   TON_FIT102_P6_TM.PRE 			:= 	3*1000;
   TON_FIT102_P6_TM.TimerEnable 	:=  HMI_FIT201.ALL AND HMI_MV201.STATUS=2 AND HMI_P206.STATUS=2;
   TONR(TON_FIT102_P6_TM);
   
   (*---------------------------------------------------------------------------------*)
   (*P201 Permissive*)
   HMI_P201.Permissive.0 	:= NOT HMI_LS201.Alarm;
   HMI_P201.Permissive.1 	:= HMI_MV201.STATUS=2;
   HMI_P201.Permissive.2 	:= HMI_FIT201.AH;
   HMI_P201.Permissive.3 	:= 1;
   HMI_P201.Permissive.4 	:= 1;
   HMI_P201.Permissive.5 	:= 1;
   HMI_P201.Permissive.6 	:= 1;
   HMI_P201.Permissive.7 	:= 1;
   HMI_P201.Permissive.8 	:= 1;
   HMI_P201.Permissive.9 	:= 1;
   HMI_P201.Permissive.10 	:= 1;
   HMI_P201.Permissive.11 	:= 1;
   HMI_P201.Permissive.12 	:= 1;
   HMI_P201.Permissive.13	:= 1;
   HMI_P201.Permissive.14	:= 1;
   HMI_P201.Permissive.15 	:= 1;
   
   HMI_P201_MSG.PERMISSIVE1 := HMI_P201.Permissive.0;
   HMI_P201_MSG.PERMISSIVE2 := HMI_P201.Permissive.1;
   HMI_P201_MSG.PERMISSIVE3 := HMI_P201.Permissive.2;
   HMI_P201_MSG.PERMISSIVE4 := 0;
   HMI_P201_MSG.PERMISSIVE5 := 0;
   
   (*P202 Permissive*)
   HMI_P202.Permissive.0 	:= NOT HMI_LS201.Alarm;
   HMI_P202.Permissive.1 	:= HMI_MV201.STATUS=2;
   HMI_P202.Permissive.2 	:= HMI_FIT201.AH;
   HMI_P202.Permissive.3 	:= 1;
   HMI_P202.Permissive.4 	:= 1;
   HMI_P202.Permissive.5 	:= 1;
   HMI_P202.Permissive.6 	:= 1;
   HMI_P202.Permissive.7 	:= 1;
   HMI_P202.Permissive.8 	:= 1;
   HMI_P202.Permissive.9 	:= 1;
   HMI_P202.Permissive.10 	:= 1;
   HMI_P202.Permissive.11 	:= 1;
   HMI_P202.Permissive.12 	:= 1;
   HMI_P202.Permissive.13	:= 1;
   HMI_P202.Permissive.14	:= 1;
   HMI_P202.Permissive.15 	:= 1;
   
   HMI_P202_MSG.PERMISSIVE1 := HMI_P202.Permissive.0;
   HMI_P202_MSG.PERMISSIVE2 := HMI_P202.Permissive.1;
   HMI_P202_MSG.PERMISSIVE3 := HMI_P202.Permissive.2;
   HMI_P202_MSG.PERMISSIVE4 := 0;
   HMI_P202_MSG.PERMISSIVE5 := 0;
   
   (*P203 Permissive*)
   HMI_P203.Permissive.0 	:= NOT HMI_LS202.Alarm;
   HMI_P203.Permissive.1 	:= HMI_MV201.STATUS=2;
   HMI_P203.Permissive.2 	:= HMI_FIT201.AH;
   HMI_P203.Permissive.3 	:= 1;
   HMI_P203.Permissive.4 	:= 1;
   HMI_P203.Permissive.5 	:= 1;
   HMI_P203.Permissive.6 	:= 1;
   HMI_P203.Permissive.7 	:= 1;
   HMI_P203.Permissive.8 	:= 1;
   HMI_P203.Permissive.9 	:= 1;
   HMI_P203.Permissive.10 	:= 1;
   HMI_P203.Permissive.11 	:= 1;
   HMI_P203.Permissive.12 	:= 1;
   HMI_P203.Permissive.13	:= 1;
   HMI_P203.Permissive.14	:= 1;
   HMI_P203.Permissive.15 	:= 1;
   
   HMI_P203_MSG.PERMISSIVE1 := HMI_P203.Permissive.0;
   HMI_P203_MSG.PERMISSIVE2 := HMI_P203.Permissive.1;
   HMI_P203_MSG.PERMISSIVE3 := HMI_P203.Permissive.2;
   HMI_P203_MSG.PERMISSIVE4 := 0;
   HMI_P203_MSG.PERMISSIVE5 := 0;
   
   (*P204 Permissive*)
   HMI_P204.Permissive.0 	:= NOT HMI_LS202.Alarm;
   HMI_P204.Permissive.1 	:= HMI_MV201.STATUS=2;
   HMI_P204.Permissive.2 	:= HMI_FIT201.AH;
   HMI_P204.Permissive.3 	:= 1;
   HMI_P204.Permissive.4 	:= 1;
   HMI_P204.Permissive.5 	:= 1;
   HMI_P204.Permissive.6 	:= 1;
   HMI_P204.Permissive.7 	:= 1;
   HMI_P204.Permissive.8 	:= 1;
   HMI_P204.Permissive.9 	:= 1;
   HMI_P204.Permissive.10 	:= 1;
   HMI_P204.Permissive.11 	:= 1;
   HMI_P204.Permissive.12 	:= 1;
   HMI_P204.Permissive.13	:= 1;
   HMI_P204.Permissive.14	:= 1;
   HMI_P204.Permissive.15 	:= 1;
   
   HMI_P204_MSG.PERMISSIVE1 := HMI_P204.Permissive.0;
   HMI_P204_MSG.PERMISSIVE2 := HMI_P204.Permissive.1;
   HMI_P204_MSG.PERMISSIVE3 := HMI_P204.Permissive.2;
   HMI_P204_MSG.PERMISSIVE4 := 0;
   HMI_P204_MSG.PERMISSIVE5 := 0;
   
   (*P205 Permissive*)
   HMI_P205.Permissive.0 	:= NOT HMI_LSL203.Alarm;
   HMI_P205.Permissive.1 	:= HMI_MV201.STATUS=2;
   HMI_P205.Permissive.2 	:= HMI_FIT201.AH;
   HMI_P205.Permissive.3 	:= 1;
   HMI_P205.Permissive.4 	:= 1;
   HMI_P205.Permissive.5 	:= 1;
   HMI_P205.Permissive.6 	:= 1;
   HMI_P205.Permissive.7 	:= 1;
   HMI_P205.Permissive.8 	:= 1;
   HMI_P205.Permissive.9 	:= 1;
   HMI_P205.Permissive.10 	:= 1;
   HMI_P205.Permissive.11 	:= 1;
   HMI_P205.Permissive.12 	:= 1;
   HMI_P205.Permissive.13	:= 1;
   HMI_P205.Permissive.14	:= 1;
   HMI_P205.Permissive.15 	:= 1;
   
   HMI_P205_MSG.PERMISSIVE1 := HMI_P205.Permissive.0;
   HMI_P205_MSG.PERMISSIVE2 := HMI_P205.Permissive.1;
   HMI_P205_MSG.PERMISSIVE3 := HMI_P205.Permissive.2;
   HMI_P205_MSG.PERMISSIVE4 := 0;
   HMI_P205_MSG.PERMISSIVE5 := 0;
   
   (*P206 Permissive*)
   HMI_P206.Permissive.0 	:= NOT HMI_LSL203.Alarm;
   HMI_P206.Permissive.1 	:= HMI_MV201.STATUS=2;
   HMI_P206.Permissive.2 	:= HMI_FIT201.AH;
   HMI_P206.Permissive.3 	:= 1;
   HMI_P206.Permissive.4 	:= 1;
   HMI_P206.Permissive.5 	:= 1;
   HMI_P206.Permissive.6 	:= 1;
   HMI_P206.Permissive.7 	:= 1;
   HMI_P206.Permissive.8 	:= 1;
   HMI_P206.Permissive.9 	:= 1;
   HMI_P206.Permissive.10 	:= 1;
   HMI_P206.Permissive.11 	:= 1;
   HMI_P206.Permissive.12 	:= 1;
   HMI_P206.Permissive.13	:= 1;
   HMI_P206.Permissive.14	:= 1;
   HMI_P206.Permissive.15 	:= 1;
   
   HMI_P206_MSG.PERMISSIVE1 := HMI_P206.Permissive.0;
   HMI_P206_MSG.PERMISSIVE2 := HMI_P206.Permissive.1;
   HMI_P206_MSG.PERMISSIVE3 := HMI_P206.Permissive.2;
   HMI_P206_MSG.PERMISSIVE4 := 0;
   HMI_P206_MSG.PERMISSIVE5 := 0;
   
   (*P207 Permissive*)
   HMI_P207.Permissive.0 	:= NOT HMI_LSL203.Alarm;
   HMI_P207.Permissive.1 	:= HMI_MV301.STATUS=2;
   HMI_P207.Permissive.2 	:= 1;
   HMI_P207.Permissive.3 	:= 1;
   HMI_P207.Permissive.4 	:= 1;
   HMI_P207.Permissive.5 	:= 1;
   HMI_P207.Permissive.6 	:= 1;
   HMI_P207.Permissive.7 	:= 1;
   HMI_P207.Permissive.8 	:= 1;
   HMI_P207.Permissive.9 	:= 1;
   HMI_P207.Permissive.10 	:= 1;
   HMI_P207.Permissive.11 	:= 1;
   HMI_P207.Permissive.12 	:= 1;
   HMI_P207.Permissive.13	:= 1;
   HMI_P207.Permissive.14	:= 1;
   HMI_P207.Permissive.15 	:= 1;
   
   HMI_P207_MSG.PERMISSIVE1 := HMI_P207.Permissive.0;
   HMI_P207_MSG.PERMISSIVE2 := HMI_P207.Permissive.1;
   HMI_P207_MSG.PERMISSIVE3 := HMI_P207.Permissive.2;
   HMI_P207_MSG.PERMISSIVE4 := 0;
   HMI_P207_MSG.PERMISSIVE5 := 0;
   
   (*P208 Permissive*)
   HMI_P208.Permissive.0 	:= NOT HMI_LSL203.Alarm;
   HMI_P208.Permissive.1 	:= HMI_MV301.STATUS=2;
   HMI_P208.Permissive.2 	:= 1;
   HMI_P208.Permissive.3 	:= 1;
   HMI_P208.Permissive.4 	:= 1;
   HMI_P208.Permissive.5 	:= 1;
   HMI_P208.Permissive.6 	:= 1;
   HMI_P208.Permissive.7 	:= 1;
   HMI_P208.Permissive.8 	:= 1;
   HMI_P208.Permissive.9 	:= 1;
   HMI_P208.Permissive.10 	:= 1;
   HMI_P208.Permissive.11 	:= 1;
   HMI_P208.Permissive.12 	:= 1;
   HMI_P208.Permissive.13	:= 1;
   HMI_P208.Permissive.14	:= 1;
   HMI_P208.Permissive.15 	:= 1;
   
   HMI_P208_MSG.PERMISSIVE1 := HMI_P208.Permissive.0;
   HMI_P208_MSG.PERMISSIVE2 := HMI_P208.Permissive.1;
   HMI_P208_MSG.PERMISSIVE3 := HMI_P208.Permissive.2;
   HMI_P208_MSG.PERMISSIVE4 := 0;
   HMI_P208_MSG.PERMISSIVE5 := 0;
   
   (*-------------------------------------------------------------------------------------*)
   (*P201 Shutdown*)
   HMI_P201.SD.0 	:= HMI_LS201.Alarm;
   HMI_P201.SD.1 	:= HMI_P201.STATUS=2 AND HMI_MV201.STATUS<>2;
   HMI_P201.SD.2 	:= TON_FIT102_P1_TM.DN;
   HMI_P201.SD.3 	:= 0;
   HMI_P201.SD.4 	:= 0;
   HMI_P201.SD.5 	:= 0;
   HMI_P201.SD.6 	:= 0;
   HMI_P201.SD.7 	:= 0;
   HMI_P201.SD.8 	:= 0;
   HMI_P201.SD.9 	:= 0;
   HMI_P201.SD.10 	:= 0;
   HMI_P201.SD.11 	:= 0;
   HMI_P201.SD.12 	:= 0;
   HMI_P201.SD.13 	:= 0;
   HMI_P201.SD.14 	:= 0;
   HMI_P201.SD.15 	:= 0;
   
   HMI_P201_MSG.SHUTDOWN1 := HMI_P201.SHUTDOWN.0 ;
   HMI_P201_MSG.SHUTDOWN2 := HMI_P201.SHUTDOWN.1 ;
   HMI_P201_MSG.SHUTDOWN3 := HMI_P201.SHUTDOWN.2 ;
   HMI_P201_MSG.SHUTDOWN4 := 0;
   HMI_P201_MSG.SHUTDOWN5 := 0;
   
   (*P202 Shutdown*)
   HMI_P202.SD.0 	:= HMI_LS201.Alarm;
   HMI_P202.SD.1 	:= HMI_P201.STATUS=2 AND HMI_MV201.STATUS<>2;
   HMI_P202.SD.2 	:= TON_FIT102_P2_TM.DN;
   HMI_P202.SD.3 	:= 0;
   HMI_P202.SD.4 	:= 0;
   HMI_P202.SD.5 	:= 0;
   HMI_P202.SD.6 	:= 0;
   HMI_P202.SD.7 	:= 0;
   HMI_P202.SD.8 	:= 0;
   HMI_P202.SD.9 	:= 0;
   HMI_P202.SD.10 	:= 0;
   HMI_P202.SD.11 	:= 0;
   HMI_P202.SD.12 	:= 0;
   HMI_P202.SD.13 	:= 0;
   HMI_P202.SD.14 	:= 0;
   HMI_P202.SD.15 	:= 0;
   
   HMI_P202_MSG.SHUTDOWN1 := HMI_P202.SHUTDOWN.0 ;
   HMI_P202_MSG.SHUTDOWN2 := HMI_P202.SHUTDOWN.1 ;
   HMI_P202_MSG.SHUTDOWN3 := HMI_P202.SHUTDOWN.2 ;
   HMI_P202_MSG.SHUTDOWN4 := 0;
   HMI_P202_MSG.SHUTDOWN5 := 0;
   
   (*P203 Shutdown*)
   HMI_P203.SD.0 	:= HMI_LS202.Alarm;
   HMI_P203.SD.1 	:= HMI_P201.STATUS=2 AND HMI_MV201.STATUS<>2;
   HMI_P203.SD.2 	:= TON_FIT102_P3_TM.DN;
   HMI_P203.SD.3 	:= 0;
   HMI_P203.SD.4 	:= 0;
   HMI_P203.SD.5 	:= 0;
   HMI_P203.SD.6 	:= 0;
   HMI_P203.SD.7 	:= 0;
   HMI_P203.SD.8 	:= 0;
   HMI_P203.SD.9 	:= 0;
   HMI_P203.SD.10 	:= 0;
   HMI_P203.SD.11 	:= 0;
   HMI_P203.SD.12 	:= 0;
   HMI_P203.SD.13 	:= 0;
   HMI_P203.SD.14 	:= 0;
   HMI_P203.SD.15 	:= 0;
   
   HMI_P203_MSG.SHUTDOWN1 := HMI_P203.SHUTDOWN.0 ;
   HMI_P203_MSG.SHUTDOWN2 := HMI_P203.SHUTDOWN.1 ;
   HMI_P203_MSG.SHUTDOWN3 := HMI_P203.SHUTDOWN.2 ;
   HMI_P203_MSG.SHUTDOWN4 := 0;
   HMI_P203_MSG.SHUTDOWN5 := 0;
   
   (*P204 Shutdown*)
   HMI_P204.SD.0 	:= HMI_LS202.Alarm;
   HMI_P204.SD.1 	:= HMI_P201.STATUS=2 AND HMI_MV201.STATUS<>2;
   HMI_P204.SD.2 	:= TON_FIT102_P4_TM.DN;
   HMI_P204.SD.3 	:= 0;
   HMI_P204.SD.4 	:= 0;
   HMI_P204.SD.5 	:= 0;
   HMI_P204.SD.6 	:= 0;
   HMI_P204.SD.7 	:= 0;
   HMI_P204.SD.8 	:= 0;
   HMI_P204.SD.9 	:= 0;
   HMI_P204.SD.10 	:= 0;
   HMI_P204.SD.11 	:= 0;
   HMI_P204.SD.12 	:= 0;
   HMI_P204.SD.13 	:= 0;
   HMI_P204.SD.14 	:= 0;
   HMI_P204.SD.15 	:= 0;
   
   HMI_P204_MSG.SHUTDOWN1 := HMI_P204.SHUTDOWN.0 ;
   HMI_P204_MSG.SHUTDOWN2 := HMI_P204.SHUTDOWN.1 ;
   HMI_P204_MSG.SHUTDOWN3 := HMI_P204.SHUTDOWN.2 ;
   HMI_P204_MSG.SHUTDOWN4 := 0;
   HMI_P204_MSG.SHUTDOWN5 := 0;
   
   (*P205 Shutdown*)
   HMI_P205.SD.0 	:= HMI_LSL203.Alarm;
   HMI_P205.SD.1 	:= HMI_P201.STATUS=2 AND HMI_MV201.STATUS<>2;
   HMI_P205.SD.2 	:= TON_FIT102_P5_TM.DN;
   HMI_P205.SD.3 	:= 0;
   HMI_P205.SD.4 	:= 0;
   HMI_P205.SD.5 	:= 0;
   HMI_P205.SD.6 	:= 0;
   HMI_P205.SD.7 	:= 0;
   HMI_P205.SD.8 	:= 0;
   HMI_P205.SD.9 	:= 0;
   HMI_P205.SD.10 	:= 0;
   HMI_P205.SD.11 	:= 0;
   HMI_P205.SD.12 	:= 0;
   HMI_P205.SD.13 	:= 0;
   HMI_P205.SD.14 	:= 0;
   HMI_P205.SD.15 	:= 0;
   
   HMI_P205_MSG.SHUTDOWN1 := HMI_P205.SHUTDOWN.0 ;
   HMI_P205_MSG.SHUTDOWN2 := HMI_P205.SHUTDOWN.1 ;
   HMI_P205_MSG.SHUTDOWN3 := HMI_P205.SHUTDOWN.2 ;
   HMI_P205_MSG.SHUTDOWN4 := 0;
   HMI_P205_MSG.SHUTDOWN5 := 0;
   
   (*P206 Shutdown*)
   HMI_P206.SD.0 	:= HMI_LSL203.Alarm;
   HMI_P206.SD.1 	:= HMI_P201.STATUS=2 AND HMI_MV201.STATUS<>2;
   HMI_P206.SD.2 	:= TON_FIT102_P6_TM.DN;
   HMI_P206.SD.3 	:= 0;
   HMI_P206.SD.4 	:= 0;
   HMI_P206.SD.5 	:= 0;
   HMI_P206.SD.6 	:= 0;
   HMI_P206.SD.7 	:= 0;
   HMI_P206.SD.8 	:= 0;
   HMI_P206.SD.9 	:= 0;
   HMI_P206.SD.10 	:= 0;
   HMI_P206.SD.11 	:= 0;
   HMI_P206.SD.12 	:= 0;
   HMI_P206.SD.13 	:= 0;
   HMI_P206.SD.14 	:= 0;
   HMI_P206.SD.15 	:= 0;
   
   HMI_P206_MSG.SHUTDOWN1 := HMI_P206.SHUTDOWN.0 ;
   HMI_P206_MSG.SHUTDOWN2 := HMI_P206.SHUTDOWN.1 ;
   HMI_P206_MSG.SHUTDOWN3 := HMI_P206.SHUTDOWN.2 ;
   HMI_P206_MSG.SHUTDOWN4 := 0;
   HMI_P206_MSG.SHUTDOWN5 := 0;
   
   (*P207 Shutdown*)
   HMI_P207.SD.0 	:= HMI_LSL203.Alarm;
   HMI_P207.SD.1 	:= HMI_P207.STATUS=2 AND HMI_MV301.STATUS<>2;
   HMI_P207.SD.2 	:= 0;
   HMI_P207.SD.3 	:= 0;
   HMI_P207.SD.4 	:= 0;
   HMI_P207.SD.5 	:= 0;
   HMI_P207.SD.6 	:= 0;
   HMI_P207.SD.7 	:= 0;
   HMI_P207.SD.8 	:= 0;
   HMI_P207.SD.9 	:= 0;
   HMI_P207.SD.10 	:= 0;
   HMI_P207.SD.11 	:= 0;
   HMI_P207.SD.12 	:= 0;
   HMI_P207.SD.13 	:= 0;
   HMI_P207.SD.14 	:= 0;
   HMI_P207.SD.15 	:= 0;
   
   HMI_P207_MSG.SHUTDOWN1 := HMI_P207.SHUTDOWN.0 ;
   HMI_P207_MSG.SHUTDOWN2 := HMI_P207.SHUTDOWN.1 ;
   HMI_P207_MSG.SHUTDOWN3 := 0;
   HMI_P207_MSG.SHUTDOWN4 := 0;
   HMI_P207_MSG.SHUTDOWN5 := 0;
   
   (*P208 Shutdown*)
   HMI_P208.SD.0 	:= HMI_LSL203.Alarm;
   HMI_P208.SD.1 	:= HMI_P207.STATUS=2 AND HMI_MV301.STATUS<>2;
   HMI_P208.SD.2 	:= 0;
   HMI_P208.SD.3 	:= 0;
   HMI_P208.SD.4 	:= 0;
   HMI_P208.SD.5 	:= 0;
   HMI_P208.SD.6 	:= 0;
   HMI_P208.SD.7 	:= 0;
   HMI_P208.SD.8 	:= 0;
   HMI_P208.SD.9 	:= 0;
   HMI_P208.SD.10 	:= 0;
   HMI_P208.SD.11 	:= 0;
   HMI_P208.SD.12 	:= 0;
   HMI_P208.SD.13 	:= 0;
   HMI_P208.SD.14 	:= 0;
   HMI_P208.SD.15 	:= 0;
   
   HMI_P208_MSG.SHUTDOWN1 := HMI_P208.SHUTDOWN.0 ;
   HMI_P208_MSG.SHUTDOWN2 := HMI_P208.SHUTDOWN.1 ;
   HMI_P208_MSG.SHUTDOWN3 := 0;
   HMI_P208_MSG.SHUTDOWN4 := 0;
   HMI_P208_MSG.SHUTDOWN5 := 0;
   
END_ROUTINE

ROUTINE UF_Feed   (* function block diagram *)
   SHEET 1
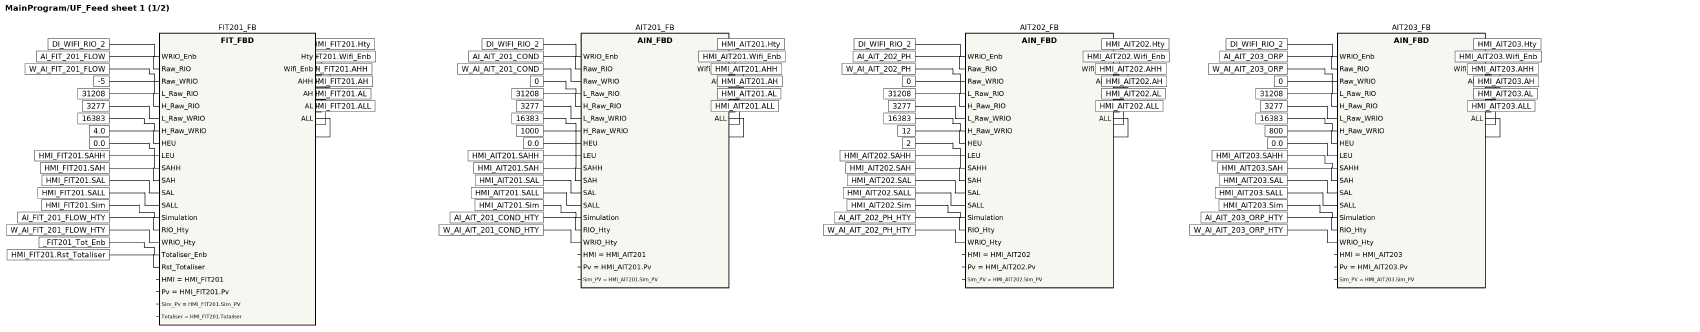
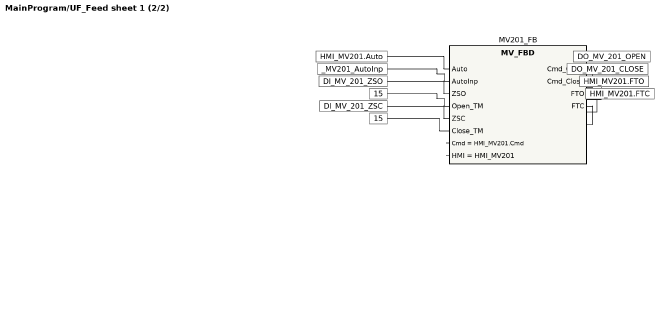
   FIT201_FB : FIT_FBD(WRIO_Enb := DI_WIFI_RIO_2, Raw_RIO := AI_FIT_201_FLOW, Raw_WRIO := W_AI_FIT_201_FLOW, L_Raw_RIO := -5, H_Raw_RIO := 31208, L_Raw_WRIO := 3277, H_Raw_WRIO := 16383, HEU := 4.0, LEU := 0.0, SAHH := HMI_FIT201.SAHH, SAH := HMI_FIT201.SAH, SAL := HMI_FIT201.SAL, SALL := HMI_FIT201.SALL, Simulation := HMI_FIT201.Sim, RIO_Hty := AI_FIT_201_FLOW_HTY, WRIO_Hty := W_AI_FIT_201_FLOW_HTY, Totaliser_Enb := _FIT201_Tot_Enb, Rst_Totaliser := HMI_FIT201.Rst_Totaliser, HMI := HMI_FIT201, Pv := HMI_FIT201.Pv, Sim_Pv := HMI_FIT201.Sim_PV, Totaliser := HMI_FIT201.Totaliser);
   HMI_FIT201.Wifi_Enb := FIT201_FB.Wifi_Enb;
   HMI_FIT201.AHH := FIT201_FB.AHH;
   HMI_FIT201.Hty := FIT201_FB.Hty;
   HMI_FIT201.AH := FIT201_FB.AH;
   HMI_FIT201.AL := FIT201_FB.AL;
   HMI_FIT201.ALL := FIT201_FB.ALL;
   AIT201_FB : AIN_FBD(WRIO_Enb := DI_WIFI_RIO_2, Raw_RIO := AI_AIT_201_COND, Raw_WRIO := W_AI_AIT_201_COND, L_Raw_RIO := 0, H_Raw_RIO := 31208, L_Raw_WRIO := 3277, H_Raw_WRIO := 16383, HEU := 1000, LEU := 0.0, SAHH := HMI_AIT201.SAHH, SAH := HMI_AIT201.SAH, SAL := HMI_AIT201.SAL, SALL := HMI_AIT201.SALL, Simulation := HMI_AIT201.Sim, RIO_Hty := AI_AIT_201_COND_HTY, WRIO_Hty := W_AI_AIT_201_COND_HTY, HMI := HMI_AIT201, Pv := HMI_AIT201.Pv, Sim_PV := HMI_AIT201.Sim_PV);
   HMI_AIT201.Wifi_Enb := AIT201_FB.Wifi_Enb;
   HMI_AIT201.AHH := AIT201_FB.AHH;
   HMI_AIT201.ALL := AIT201_FB.ALL;
   HMI_AIT201.Hty := AIT201_FB.Hty;
   HMI_AIT201.AH := AIT201_FB.AH;
   HMI_AIT201.AL := AIT201_FB.AL;
   AIT202_FB : AIN_FBD(WRIO_Enb := DI_WIFI_RIO_2, Raw_RIO := AI_AIT_202_PH, Raw_WRIO := W_AI_AIT_202_PH, L_Raw_RIO := 0, H_Raw_RIO := 31208, L_Raw_WRIO := 3277, H_Raw_WRIO := 16383, HEU := 12, LEU := 2, SAHH := HMI_AIT202.SAHH, SAH := HMI_AIT202.SAH, SAL := HMI_AIT202.SAL, SALL := HMI_AIT202.SALL, Simulation := HMI_AIT202.Sim, RIO_Hty := AI_AIT_202_PH_HTY, WRIO_Hty := W_AI_AIT_202_PH_HTY, HMI := HMI_AIT202, Pv := HMI_AIT202.Pv, Sim_PV := HMI_AIT202.Sim_PV);
   HMI_AIT202.Wifi_Enb := AIT202_FB.Wifi_Enb;
   HMI_AIT202.AHH := AIT202_FB.AHH;
   HMI_AIT202.ALL := AIT202_FB.ALL;
   HMI_AIT202.Hty := AIT202_FB.Hty;
   HMI_AIT202.AH := AIT202_FB.AH;
   HMI_AIT202.AL := AIT202_FB.AL;
   AIT203_FB : AIN_FBD(WRIO_Enb := DI_WIFI_RIO_2, Raw_RIO := AI_AIT_203_ORP, Raw_WRIO := W_AI_AIT_203_ORP, L_Raw_RIO := 0, H_Raw_RIO := 31208, L_Raw_WRIO := 3277, H_Raw_WRIO := 16383, HEU := 800, LEU := 0.0, SAHH := HMI_AIT203.SAHH, SAH := HMI_AIT203.SAH, SAL := HMI_AIT203.SAL, SALL := HMI_AIT203.SALL, Simulation := HMI_AIT203.Sim, RIO_Hty := AI_AIT_203_ORP_HTY, WRIO_Hty := W_AI_AIT_203_ORP_HTY, HMI := HMI_AIT203, Pv := HMI_AIT203.Pv, Sim_PV := HMI_AIT203.Sim_PV);
   HMI_AIT203.Wifi_Enb := AIT203_FB.Wifi_Enb;
   HMI_AIT203.AHH := AIT203_FB.AHH;
   HMI_AIT203.ALL := AIT203_FB.ALL;
   HMI_AIT203.Hty := AIT203_FB.Hty;
   HMI_AIT203.AH := AIT203_FB.AH;
   HMI_AIT203.AL := AIT203_FB.AL;
   MV201_FB : MV_FBD(Auto := HMI_MV201.Auto, AutoInp := _MV201_AutoInp, ZSO := DI_MV_201_ZSO, Open_TM := 15, ZSC := DI_MV_201_ZSC, Close_TM := 15, Cmd := HMI_MV201.Cmd, HMI := HMI_MV201);
   DO_MV_201_CLOSE := MV201_FB.Cmd_Close;
   DO_MV_201_OPEN := MV201_FB.Cmd_Open;
   HMI_MV201.FTO := MV201_FB.FTO;
   HMI_MV201.FTC := MV201_FB.FTC;
END_ROUTINE

ROUTINE VALIDATE_INPUT   (* structured text *)
// VALIDATING THE STATES WITH RESPECT TO OTHER STATES
   (*SECOND PULSE*)
   
   
   
   
   
   	IF HMI_PLANT.START OR HMI_PLANT.STOP   THEN
   
   			ATTACK :=0;
   
   	END_IF;
   
   
   
   
   // NO ESTIMATION FOR LEVEL
   
   
   
   //BACKWARD CHECKING
   
   (* LIT301 LOW VALUE MV201 SHOULD BE CLOSE  *)
   IF HMI_LIT301.AL THEN
   	IF HMI_MV201.Status <> 2  THEN
   		ATTACK := 1;
   	END_IF;
   END_IF;
   
   (* LIT301 HIGH VALUE MV201 SHOULD BE CLOSE*)
   
   IF HMI_LIT301.AL THEN
   	IF HMI_MV201.Status <> 1  THEN
   		ATTACK := 1;
   	END_IF;
   END_IF;
   
   ATTACK:=0;
   
END_ROUTINE
END_PROGRAM
